    |   movel(p[0.471269, -0.071095, -0.000100, 0.000000, 3.141593, 0.000000],accel_mss,speed_ms,0,blend_radius_m)
    |   movel(p[0.470803, -0.071857, -0.000100, 0.000000, -3.141593, 0.000000],accel_mss,speed_ms,0,blend_radius_m)
    |   movel(p[0.470715, -0.072007, -0.000100, 0.000000, 3.141593, 0.000000],accel_mss,speed_ms,0,0.000)
    |   movel(p[0.470597, -0.072221, -0.000100, 0.000000, -3.141593, 0.000000],accel_mss,speed_ms,0,0.000)
    |   movel(p[0.470473, -0.072456, -0.000100, 0.000000, -3.141593, 0.000000],accel_mss,speed_ms,0,0.000)
    |   movel(p[0.470361, -0.072678, -0.000100, 0.000000, -3.141593, 0.000000],accel_mss,speed_ms,0,0.000)
    |   movel(p[0.470239, -0.072912, -0.000100, 0.000000, -3.141593, 0.000000],accel_mss,speed_ms,0,0.000)
    |   movel(p[0.470084, -0.073181, -0.000100, 0.000000, -3.141593, 0.000000],accel_mss,speed_ms,0,0.000)
    |   movel(p[0.469922, -0.073443, -0.000100, 0.000000, -3.141593, 0.000000],accel_mss,speed_ms,0,0.000)
    |   movel(p[0.469779, -0.073653, -0.000100, 0.000000, -3.141593, 0.000000],accel_mss,speed_ms,0,0.000)
    |   movel(p[0.469648, -0.073842, -0.000100, 0.000000, -3.141593, 0.000000],accel_mss,speed_ms,0,0.000)
    |   movel(p[0.469521, -0.074037, -0.000100, 0.000000, -3.141593, 0.000000],accel_mss,speed_ms,0,0.000)
    |   movel(p[0.469416, -0.074212, -0.000100, 0.000000, -3.141593, 0.000000],accel_mss,speed_ms,0,0.000)
    |   movel(p[0.469356, -0.074328, -0.000100, 0.000000, -3.141593, 0.000000],accel_mss,speed_ms,0,0.000)
    |   movel(p[0.469299, -0.074444, -0.000100, 0.000000, -3.141593, 0.000000],accel_mss,speed_ms,0,0.000)
    |   movel(p[0.469200, -0.074619, -0.000100, 0.000000, -3.141593, 0.000000],accel_mss,speed_ms,0,0.000)
    |   movel(p[0.469084, -0.074815, -0.000100, 0.000000, -3.141593, 0.000000],accel_mss,speed_ms,0,0.000)
    |   movel(p[0.468964, -0.075003, -0.000100, 0.000000, -3.141593, 0.000000],accel_mss,speed_ms,0,0.000)
    |   movel(p[0.468837, -0.075208, -0.000100, 0.000000, -3.141593, 0.000000],accel_mss,speed_ms,0,0.000)
    |   movel(p[0.468696, -0.075453, -0.000100, 0.000000, -3.141593, 0.000000],accel_mss,speed_ms,0,0.000)
    |   movel(p[0.468564, -0.075699, -0.000100, 0.000000, -3.141593, 0.000000],accel_mss,speed_ms,0,0.000)
    |   movel(p[0.468464, -0.075903, -0.000100, 0.000000, -3.141593, 0.000000],accel_mss,speed_ms,0,0.000)
    |   movel(p[0.468366, -0.076091, -0.000100, 0.000000, -3.141593, 0.000000],accel_mss,speed_ms,0,0.000)
    |   movel(p[0.468243, -0.076283, -0.000100, 0.000000, -3.141593, 0.000000],accel_mss,speed_ms,0,0.000)
    |   movel(p[0.468114, -0.076453, -0.000100, 0.000000, 3.141593, 0.000000],accel_mss,speed_ms,0,0.000)
    |   movel(p[0.468002, -0.076565, -0.000100, 0.000000, -3.141593, 0.000000],accel_mss,speed_ms,0,0.000)
    |   movel(p[0.467885, -0.076688, -0.000100, 0.000000, -3.141593, 0.000000],accel_mss,speed_ms,0,0.000)
    |   movel(p[0.467739, -0.076896, -0.000100, 0.000000, -3.141593, 0.000000],accel_mss,speed_ms,0,0.000)
    |   movel(p[0.467592, -0.077142, -0.000100, 0.000000, -3.141593, 0.000000],accel_mss,speed_ms,0,0.000)
    |   movel(p[0.467465, -0.077394, -0.000100, 0.000000, -3.141593, 0.000000],accel_mss,speed_ms,0,0.000)
    |   movel(p[0.467335, -0.077651, -0.000100, 0.000000, -3.141593, 0.000000],accel_mss,speed_ms,0,0.000)
    |   movel(p[0.467175, -0.077912, -0.000100, 0.000000, -3.141593, 0.000000],accel_mss,speed_ms,0,0.000)
    |   movel(p[0.467012, -0.078142, -0.000100, 0.000000, -3.141593, 0.000000],accel_mss,speed_ms,0,0.000)
    |   movel(p[0.466873, -0.078293, -0.000100, 0.000000, -3.141593, 0.000000],accel_mss,speed_ms,0,0.000)
    |   movel(p[0.466753, -0.078412, -0.000100, 0.000000, -3.141593, 0.000000],accel_mss,speed_ms,0,0.000)
    |   movel(p[0.466653, -0.078535, -0.000100, 0.000000, -3.141593, 0.000000],accel_mss,speed_ms,0,0.000)
    |   movel(p[0.466581, -0.078648, -0.000100, 0.000000, -3.141593, 0.000000],accel_mss,speed_ms,0,0.000)
    |   movel(p[0.466531, -0.078815, -0.000100, 0.000000, -3.141593, 0.000000],accel_mss,speed_ms,0,0.000)
    |   movel(p[0.466319, -0.079103, -0.000100, 0.000000, -3.141593, 0.000000],accel_mss,speed_ms,0,0.000)
    |   movel(p[0.466052, -0.079439, -0.000100, 0.000000, -3.141593, 0.000000],accel_mss,speed_ms,0,0.000)
    |   movel(p[0.465736, -0.079810, -0.000100, 0.000000, -3.141593, 0.000000],accel_mss,speed_ms,0,0.000)
    |   movel(p[0.465420, -0.080180, -0.000100, 0.000000, -3.141593, 0.000000],accel_mss,speed_ms,0,0.000)
    |   movel(p[0.465153, -0.080514, -0.000100, 0.000000, -3.141593, 0.000000],accel_mss,speed_ms,0,0.000)
    |   movel(p[0.464939, -0.080799, -0.000100, 0.000000, -3.141593, 0.000000],accel_mss,speed_ms,0,0.000)
    |   movel(p[0.464837, -0.081062, -0.000100, 0.000000, -3.141593, 0.000000],accel_mss,speed_ms,0,0.000)
    |   movel(p[0.464374, -0.081495, -0.000100, 0.000000, 3.141593, 0.000000],accel_mss,speed_ms,0,blend_radius_m)
    |   movel(p[0.463896, -0.081907, -0.000100, 0.000000, -3.141593, 0.000000],accel_mss,speed_ms,0,blend_radius_m)
    |   movel(p[0.463697, -0.081978, -0.000100, 0.000000, -3.141593, 0.000000],accel_mss,speed_ms,0,0.000)
    |   movel(p[0.463600, -0.082033, -0.000100, 0.000000, -3.141593, 0.000000],accel_mss,speed_ms,0,0.000)
    |   movel(p[0.463560, -0.082166, -0.000100, 0.000000, -3.141593, 0.000000],accel_mss,speed_ms,0,0.000)
    |   movel(p[0.463460, -0.082347, -0.000100, 0.000000, -3.141593, 0.000000],accel_mss,speed_ms,0,0.000)
    |   movel(p[0.463351, -0.082441, -0.000100, 0.000000, -3.141593, 0.000000],accel_mss,speed_ms,0,0.000)
    |   movel(p[0.463222, -0.082518, -0.000100, 0.000000, -3.141593, 0.000000],accel_mss,speed_ms,0,0.000)
    |   movel(p[0.463052, -0.082603, -0.000100, 0.000000, -3.141593, 0.000000],accel_mss,speed_ms,0,0.000)
    |   movel(p[0.462809, -0.082727, -0.000100, 0.000000, -3.141593, 0.000000],accel_mss,speed_ms,0,0.000)
    |   movel(p[0.462540, -0.082865, -0.000100, 0.000000, -3.141593, 0.000000],accel_mss,speed_ms,0,0.000)
    |   movel(p[0.462286, -0.082998, -0.000100, 0.000000, -3.141593, 0.000000],accel_mss,speed_ms,0,0.000)
    |   movel(p[0.460770, -0.083741, -0.000100, 0.000000, -3.141593, 0.000000],accel_mss,speed_ms,0,blend_radius_m)
    |   movel(p[0.459479, -0.084259, -0.000100, 0.000000, -3.141593, 0.000000],accel_mss,speed_ms,0,blend_radius_m)
    |   movel(p[0.458369, -0.084574, -0.000100, 0.000000, -3.141593, 0.000000],accel_mss,speed_ms,0,blend_radius_m)
    |   movel(p[0.457411, -0.084692, -0.000100, 0.000000, -3.141593, 0.000000],accel_mss,speed_ms,0,blend_radius_m)
    |   movel(p[0.457160, -0.084702, -0.000100, 0.000000, -3.141593, 0.000000],accel_mss,speed_ms,0,0.000)
    |   movel(p[0.456832, -0.084723, -0.000100, 0.000000, -3.141593, 0.000000],accel_mss,speed_ms,0,0.000)
    |   movel(p[0.456488, -0.084750, -0.000100, 0.000000, -3.141593, 0.000000],accel_mss,speed_ms,0,0.000)
    |   movel(p[0.456178, -0.084780, -0.000100, 0.000000, -3.141593, 0.000000],accel_mss,speed_ms,0,0.000)
    |   movel(p[0.455825, -0.084817, -0.000100, 0.000000, -3.141593, 0.000000],accel_mss,speed_ms,0,0.000)
    |   movel(p[0.455471, -0.084855, -0.000100, 0.000000, -3.141593, 0.000000],accel_mss,speed_ms,0,0.000)
    |   movel(p[0.455487, -0.085515, -0.000100, 0.000000, -3.141593, 0.000000],accel_mss,speed_ms,0,blend_radius_m)
    |   movel(p[0.455503, -0.086174, -0.000100, 0.000000, -3.141593, 0.000000],accel_mss,speed_ms,0,blend_radius_m)
    |   movel(p[0.455510, -0.086885, -0.000100, 0.000000, -3.141593, 0.000000],accel_mss,speed_ms,0,blend_radius_m)
    |   movel(p[0.455478, -0.087299, -0.000100, 0.000000, -3.141593, 0.000000],accel_mss,speed_ms,0,0.000)
    |   movel(p[0.455402, -0.087577, -0.000100, 0.000000, 3.141593, 0.000000],accel_mss,speed_ms,0,0.000)
    |   movel(p[0.455266, -0.087793, -0.000100, 0.000000, -3.141593, 0.000000],accel_mss,speed_ms,0,0.000)
    |   movel(p[0.454617, -0.088208, -0.000100, 0.000000, -3.141593, 0.000000],accel_mss,speed_ms,0,blend_radius_m)
    |   movel(p[0.453609, -0.088391, -0.000100, 0.000000, -3.141593, 0.000000],accel_mss,speed_ms,0,blend_radius_m)
    |   movel(p[0.452601, -0.088329, -0.000100, 0.000000, -3.141593, 0.000000],accel_mss,speed_ms,0,blend_radius_m)
    |   movel(p[0.451957, -0.087990, -0.000100, 0.000000, -3.141593, 0.000000],accel_mss,speed_ms,0,blend_radius_m)
    |   movel(p[0.451797, -0.087787, -0.000100, 0.000000, -3.141593, 0.000000],accel_mss,speed_ms,0,0.000)
    |   movel(p[0.451704, -0.087566, -0.000100, 0.000000, -3.141593, 0.000000],accel_mss,speed_ms,0,0.000)
    |   movel(p[0.451660, -0.087274, -0.000100, 0.000000, -3.141593, 0.000000],accel_mss,speed_ms,0,0.000)
    |   movel(p[0.451656, -0.086831, -0.000100, 0.000000, -3.141593, 0.000000],accel_mss,speed_ms,0,0.000)
    |   movel(p[0.451685, -0.086359, -0.000100, 0.000000, -3.141593, 0.000000],accel_mss,speed_ms,0,0.000)
    |   movel(p[0.451754, -0.086060, -0.000100, 0.000000, -3.141593, 0.000000],accel_mss,speed_ms,0,0.000)
    |   movel(p[0.451891, -0.085814, -0.000100, 0.000000, -3.141593, 0.000000],accel_mss,speed_ms,0,0.000)
    |   movel(p[0.452139, -0.085531, -0.000100, 0.000000, -3.141593, 0.000000],accel_mss,speed_ms,0,0.000)
    |   movel(p[0.452370, -0.085300, -0.000100, 0.000000, -3.141593, 0.000000],accel_mss,speed_ms,0,0.000)
    |   movel(p[0.452601, -0.085069, -0.000100, 0.000000, -3.141593, 0.000000],accel_mss,speed_ms,0,0.000)
    |   movel(p[0.452594, -0.085421, -0.000100, 0.000000, -3.141593, 0.000000],accel_mss,speed_ms,0,0.000)
    |   movel(p[0.452587, -0.085773, -0.000100, 0.000000, -3.141593, 0.000000],accel_mss,speed_ms,0,0.000)
    |   movel(p[0.452617, -0.086277, -0.000100, 0.000000, 3.141593, 0.000000],accel_mss,speed_ms,0,blend_radius_m)
    |   movel(p[0.452736, -0.086636, -0.000100, 0.000000, -3.141593, 0.000000],accel_mss,speed_ms,0,0.000)
    |   movel(p[0.452940, -0.086850, -0.000100, 0.000000, -3.141593, 0.000000],accel_mss,speed_ms,0,0.000)
    |   movel(p[0.453221, -0.086928, -0.000100, 0.000000, -3.141593, 0.000000],accel_mss,speed_ms,0,0.000)
    |   movel(p[0.453501, -0.086830, -0.000100, 0.000000, -3.141593, 0.000000],accel_mss,speed_ms,0,0.000)
    |   movel(p[0.453742, -0.086550, -0.000100, 0.000000, -3.141593, 0.000000],accel_mss,speed_ms,0,0.000)
    |   movel(p[0.453906, -0.086136, -0.000100, 0.000000, -3.141593, 0.000000],accel_mss,speed_ms,0,0.000)
    |   movel(p[0.453961, -0.085650, -0.000100, 0.000000, -3.141593, 0.000000],accel_mss,speed_ms,0,0.000)
    |   movel(p[0.453921, -0.085195, -0.000100, 0.000000, -3.141593, 0.000000],accel_mss,speed_ms,0,0.000)
    |   movel(p[0.453793, -0.084901, -0.000100, 0.000000, -3.141593, 0.000000],accel_mss,speed_ms,0,0.000)
    |   movel(p[0.453566, -0.084736, -0.000100, 0.000000, -3.141593, 0.000000],accel_mss,speed_ms,0,0.000)
    |   movel(p[0.453228, -0.084678, -0.000100, 0.000000, -3.141593, 0.000000],accel_mss,speed_ms,0,0.000)
    |   movel(p[0.452761, -0.084607, -0.000100, 0.000000, -3.141593, 0.000000],accel_mss,speed_ms,0,0.000)
    |   movel(p[0.451120, -0.084082, -0.000100, 0.000000, -3.141593, 0.000000],accel_mss,speed_ms,0,blend_radius_m)
    |   movel(p[0.449478, -0.083535, -0.000100, 0.000000, -3.141593, 0.000000],accel_mss,speed_ms,0,blend_radius_m)
    |   movel(p[0.449086, -0.083326, -0.000100, 0.000000, -3.141593, 0.000000],accel_mss,speed_ms,0,0.000)
    |   movel(p[0.448884, -0.083190, -0.000100, 0.000000, -3.141593, 0.000000],accel_mss,speed_ms,0,0.000)
    |   movel(p[0.448382, -0.082901, -0.000100, 0.000000, -3.141593, 0.000000],accel_mss,speed_ms,0,blend_radius_m)
    |   movel(p[0.447798, -0.082577, -0.000100, 0.000000, -3.141593, 0.000000],accel_mss,speed_ms,0,blend_radius_m)
    |   movel(p[0.447201, -0.082257, -0.000100, 0.000000, 3.141593, 0.000000],accel_mss,speed_ms,0,blend_radius_m)
    |   movel(p[0.446964, -0.082117, -0.000100, 0.000000, -3.141593, 0.000000],accel_mss,speed_ms,0,0.000)
    |   movel(p[0.446696, -0.081927, -0.000100, 0.000000, -3.141593, 0.000000],accel_mss,speed_ms,0,0.000)
    |   movel(p[0.446438, -0.081720, -0.000100, 0.000000, -3.141593, 0.000000],accel_mss,speed_ms,0,0.000)
    |   movel(p[0.446235, -0.081527, -0.000100, 0.000000, -3.141593, 0.000000],accel_mss,speed_ms,0,0.000)
    |   movel(p[0.446056, -0.081355, -0.000100, 0.000000, -3.141593, 0.000000],accel_mss,speed_ms,0,0.000)
    |   movel(p[0.445873, -0.081210, -0.000100, 0.000000, -3.141593, 0.000000],accel_mss,speed_ms,0,0.000)
    |   movel(p[0.445710, -0.081106, -0.000100, 0.000000, -3.141593, 0.000000],accel_mss,speed_ms,0,0.000)
    |   movel(p[0.445608, -0.081078, -0.000100, 0.000000, 3.141593, 0.000000],accel_mss,speed_ms,0,0.000)
    |   movel(p[0.445469, -0.081011, -0.000100, 0.000000, -3.141593, 0.000000],accel_mss,speed_ms,0,0.000)
    |   movel(p[0.445411, -0.080849, -0.000100, 0.000000, -3.141593, 0.000000],accel_mss,speed_ms,0,0.000)
    |   movel(p[0.445334, -0.080659, -0.000100, 0.000000, -3.141593, 0.000000],accel_mss,speed_ms,0,0.000)
    |   movel(p[0.445249, -0.080578, -0.000100, 0.000000, -3.141593, 0.000000],accel_mss,speed_ms,0,0.000)
    |   movel(p[0.445148, -0.080525, -0.000100, 0.000000, -3.141593, 0.000000],accel_mss,speed_ms,0,0.000)
    |   movel(p[0.444857, -0.080365, -0.000100, 0.000000, -3.141593, 0.000000],accel_mss,speed_ms,0,0.000)
    |   movel(p[0.444481, -0.080040, -0.000100, 0.000000, -3.141593, 0.000000],accel_mss,speed_ms,0,0.000)
    |   movel(p[0.444144, -0.079691, -0.000100, 0.000000, -3.141593, 0.000000],accel_mss,speed_ms,0,0.000)
    |   movel(p[0.444065, -0.079492, -0.000100, 0.000000, -3.141593, 0.000000],accel_mss,speed_ms,0,0.000)
    |   movel(p[0.443947, -0.079271, -0.000100, 0.000000, 3.141593, 0.000000],accel_mss,speed_ms,0,0.000)
    |   movel(p[0.443820, -0.079118, -0.000100, 0.000000, -3.141593, 0.000000],accel_mss,speed_ms,0,0.000)
    |   movel(p[0.443670, -0.078967, -0.000100, 0.000000, 3.141593, 0.000000],accel_mss,speed_ms,0,0.000)
    |   movel(p[0.443510, -0.078806, -0.000100, 0.000000, -3.141593, 0.000000],accel_mss,speed_ms,0,0.000)
    |   movel(p[0.443354, -0.078622, -0.000100, 0.000000, 3.141593, 0.000000],accel_mss,speed_ms,0,0.000)
    |   movel(p[0.443222, -0.078444, -0.000100, 0.000000, -3.141593, 0.000000],accel_mss,speed_ms,0,0.000)
    |   movel(p[0.443143, -0.078303, -0.000100, 0.000000, 3.141593, 0.000000],accel_mss,speed_ms,0,0.000)
    |   movel(p[0.443060, -0.078131, -0.000100, 0.000000, -3.141593, 0.000000],accel_mss,speed_ms,0,0.000)
    |   movel(p[0.442893, -0.077805, -0.000100, 0.000000, -3.141593, 0.000000],accel_mss,speed_ms,0,0.000)
    |   movel(p[0.442694, -0.077424, -0.000100, 0.000000, -3.141593, 0.000000],accel_mss,speed_ms,0,0.000)
    |   movel(p[0.442484, -0.077028, -0.000100, 0.000000, 3.141593, 0.000000],accel_mss,speed_ms,0,0.000)
    |   movel(p[0.442106, -0.076250, -0.000100, 0.000000, -3.141593, 0.000000],accel_mss,speed_ms,0,blend_radius_m)
    |   movel(p[0.441737, -0.075346, -0.000100, 0.000000, -3.141593, 0.000000],accel_mss,speed_ms,0,blend_radius_m)
    |   movel(p[0.441438, -0.074482, -0.000100, 0.000000, 3.141593, 0.000000],accel_mss,speed_ms,0,blend_radius_m)
    |   movel(p[0.441290, -0.073856, -0.000100, 0.000000, -3.141593, 0.000000],accel_mss,speed_ms,0,blend_radius_m)
    |   movel(p[0.441095, -0.072461, -0.000100, 0.000000, -3.141593, 0.000000],accel_mss,speed_ms,0,blend_radius_m)
    |   movel(p[0.440999, -0.071329, -0.000100, 0.000000, -3.141593, 0.000000],accel_mss,speed_ms,0,blend_radius_m)
    |   movel(p[0.440988, -0.070256, -0.000100, 0.000000, 3.141593, 0.000000],accel_mss,speed_ms,0,blend_radius_m)
    |   movel(p[0.441055, -0.069048, -0.000100, 0.000000, -3.141593, 0.000000],accel_mss,speed_ms,0,blend_radius_m)
    |   movel(p[0.441120, -0.068309, -0.000100, 0.000000, -3.141593, 0.000000],accel_mss,speed_ms,0,blend_radius_m)
    |   movel(p[0.441186, -0.067613, -0.000100, 0.000000, 3.141593, 0.000000],accel_mss,speed_ms,0,blend_radius_m)
    |   movel(p[0.441247, -0.067027, -0.000100, 0.000000, -3.141593, 0.000000],accel_mss,speed_ms,0,blend_radius_m)
    |   movel(p[0.441285, -0.066753, -0.000100, 0.000000, -3.141593, 0.000000],accel_mss,speed_ms,0,0.000)
    |   movel(p[0.441320, -0.066543, -0.000100, 0.000000, -3.141593, 0.000000],accel_mss,speed_ms,0,0.000)
    |   movel(p[0.441364, -0.066281, -0.000100, 0.000000, -3.141593, 0.000000],accel_mss,speed_ms,0,0.000)
    |   movel(p[0.441408, -0.066012, -0.000100, 0.000000, 3.141593, 0.000000],accel_mss,speed_ms,0,0.000)
    |   movel(p[0.441447, -0.065778, -0.000100, 0.000000, -3.141593, 0.000000],accel_mss,speed_ms,0,0.000)
    |   movel(p[0.441556, -0.065265, -0.000100, 0.000000, 3.141593, 0.000000],accel_mss,speed_ms,0,blend_radius_m)
    |   movel(p[0.441750, -0.064582, -0.000100, 0.000000, -3.141593, 0.000000],accel_mss,speed_ms,0,blend_radius_m)
    |   movel(p[0.441982, -0.063877, -0.000100, 0.000000, -3.141593, 0.000000],accel_mss,speed_ms,0,blend_radius_m)
    |   movel(p[0.442212, -0.063281, -0.000100, 0.000000, -3.141593, 0.000000],accel_mss,speed_ms,0,blend_radius_m)
    |   movel(p[0.442288, -0.063093, -0.000100, 0.000000, -3.141593, 0.000000],accel_mss,speed_ms,0,0.000)
    |   movel(p[0.442352, -0.062922, -0.000100, 0.000000, -3.141593, 0.000000],accel_mss,speed_ms,0,0.000)
    |   movel(p[0.442402, -0.062777, -0.000100, 0.000000, -3.141593, 0.000000],accel_mss,speed_ms,0,0.000)
    |   movel(p[0.442467, -0.062473, -0.000100, 0.000000, -3.141593, 0.000000],accel_mss,speed_ms,0,0.000)
    |   movel(p[0.442814, -0.061765, -0.000100, 0.000000, -3.141593, 0.000000],accel_mss,speed_ms,0,blend_radius_m)
    |   movel(p[0.443178, -0.061071, -0.000100, 0.000000, 3.141593, 0.000000],accel_mss,speed_ms,0,blend_radius_m)
    |   movel(p[0.443358, -0.060852, -0.000100, 0.000000, -3.141593, 0.000000],accel_mss,speed_ms,0,0.000)
    |   movel(p[0.443674, -0.060687, -0.000100, 0.000000, -3.141593, 0.000000],accel_mss,speed_ms,0,0.000)
    |   movel(p[0.444303, -0.060542, -0.000100, 0.000000, -3.141593, 0.000000],accel_mss,speed_ms,0,blend_radius_m)
    |   movel(p[0.444942, -0.060444, -0.000100, 0.000000, -3.141593, 0.000000],accel_mss,speed_ms,0,blend_radius_m)
    |   movel(p[0.445156, -0.060516, -0.000100, 0.000000, 3.141593, 0.000000],accel_mss,speed_ms,0,0.000)
    |   movel(p[0.445177, -0.060614, -0.000100, 0.000000, -3.141593, 0.000000],accel_mss,speed_ms,0,0.000)
    |   movel(p[0.444985, -0.061101, -0.000100, 0.000000, -3.141593, 0.000000],accel_mss,speed_ms,0,blend_radius_m)
    |   movel(p[0.444730, -0.061679, -0.000100, 0.000000, -3.141593, 0.000000],accel_mss,speed_ms,0,blend_radius_m)
    |   movel(p[0.444406, -0.062343, -0.000100, 0.000000, -3.141593, 0.000000],accel_mss,speed_ms,0,blend_radius_m)
    |   movel(p[0.443971, -0.063198, -0.000100, 0.000000, 3.141593, 0.000000],accel_mss,speed_ms,0,blend_radius_m)
    |   movel(p[0.443536, -0.064053, -0.000100, 0.000000, -3.141593, 0.000000],accel_mss,speed_ms,0,blend_radius_m)
    |   movel(p[0.443521, -0.065328, -0.000100, 0.000000, -3.141593, 0.000000],accel_mss,speed_ms,0,blend_radius_m)
    |   movel(p[0.443507, -0.066603, -0.000100, 0.000000, -3.141593, 0.000000],accel_mss,speed_ms,0,blend_radius_m)
    |   movel(p[0.443507, -0.067635, -0.000100, 0.000000, 3.141593, 0.000000],accel_mss,speed_ms,0,blend_radius_m)
    |   movel(p[0.443532, -0.068625, -0.000100, 0.000000, 3.141593, 0.000000],accel_mss,speed_ms,0,blend_radius_m)
    |   movel(p[0.443574, -0.069465, -0.000100, 0.000000, -3.141593, 0.000000],accel_mss,speed_ms,0,blend_radius_m)
    |   movel(p[0.443632, -0.069903, -0.000100, 0.000000, 3.141593, 0.000000],accel_mss,speed_ms,0,0.000)
    |   movel(p[0.444078, -0.071666, -0.000100, 0.000000, -3.141593, 0.000000],accel_mss,speed_ms,0,blend_radius_m)
    |   movel(p[0.444658, -0.073264, -0.000100, 0.000000, -3.141593, 0.000000],accel_mss,speed_ms,0,blend_radius_m)
    |   movel(p[0.445338, -0.074619, -0.000100, 0.000000, 3.141593, 0.000000],accel_mss,speed_ms,0,blend_radius_m)
    |   movel(p[0.446084, -0.075645, -0.000100, 0.000000, -3.141593, 0.000000],accel_mss,speed_ms,0,blend_radius_m)
    |   movel(p[0.446343, -0.075942, -0.000100, 0.000000, -3.141593, 0.000000],accel_mss,speed_ms,0,0.000)
    |   movel(p[0.446562, -0.076211, -0.000100, 0.000000, -3.141593, 0.000000],accel_mss,speed_ms,0,0.000)
    |   movel(p[0.446737, -0.076442, -0.000100, 0.000000, -3.141593, 0.000000],accel_mss,speed_ms,0,0.000)
    |   movel(p[0.446821, -0.076682, -0.000100, 0.000000, -3.141593, 0.000000],accel_mss,speed_ms,0,0.000)
    |   movel(p[0.447095, -0.076986, -0.000100, 0.000000, -3.141593, 0.000000],accel_mss,speed_ms,0,0.000)
    |   movel(p[0.447392, -0.077267, -0.000100, 0.000000, -3.141593, 0.000000],accel_mss,speed_ms,0,0.000)
    |   movel(p[0.447554, -0.077328, -0.000100, 0.000000, -3.141593, 0.000000],accel_mss,speed_ms,0,0.000)
    |   movel(p[0.447902, -0.077540, -0.000100, 0.000000, -3.141593, 0.000000],accel_mss,speed_ms,0,0.000)
    |   movel(p[0.448206, -0.077774, -0.000100, 0.000000, -3.141593, 0.000000],accel_mss,speed_ms,0,0.000)
    |   movel(p[0.448541, -0.078051, -0.000100, 0.000000, -3.141593, 0.000000],accel_mss,speed_ms,0,0.000)
    |   movel(p[0.448908, -0.078346, -0.000100, 0.000000, -3.141593, 0.000000],accel_mss,speed_ms,0,0.000)
    |   movel(p[0.449314, -0.078637, -0.000100, 0.000000, -3.141593, 0.000000],accel_mss,speed_ms,0,0.000)
    |   movel(p[0.449697, -0.078884, -0.000100, 0.000000, -3.141593, 0.000000],accel_mss,speed_ms,0,0.000)
    |   movel(p[0.449986, -0.079033, -0.000100, 0.000000, -3.141593, 0.000000],accel_mss,speed_ms,0,0.000)
    |   movel(p[0.450235, -0.079143, -0.000100, 0.000000, -3.141593, 0.000000],accel_mss,speed_ms,0,0.000)
    |   movel(p[0.450487, -0.079258, -0.000100, 0.000000, -3.141593, 0.000000],accel_mss,speed_ms,0,0.000)
    |   movel(p[0.450708, -0.079364, -0.000100, 0.000000, -3.141593, 0.000000],accel_mss,speed_ms,0,0.000)
    |   movel(p[0.450848, -0.079436, -0.000100, 0.000000, -3.141593, 0.000000],accel_mss,speed_ms,0,0.000)
    |   movel(p[0.451298, -0.079673, -0.000100, 0.000000, -3.141593, 0.000000],accel_mss,speed_ms,0,blend_radius_m)
    |   movel(p[0.451639, -0.079837, -0.000100, 0.000000, 3.141593, 0.000000],accel_mss,speed_ms,0,0.000)
    |   movel(p[0.452020, -0.079998, -0.000100, 0.000000, -3.141593, 0.000000],accel_mss,speed_ms,0,0.000)
    |   movel(p[0.452633, -0.080235, -0.000100, 0.000000, -3.141593, 0.000000],accel_mss,speed_ms,0,blend_radius_m)
    |   movel(p[0.454596, -0.080839, -0.000100, 0.000000, -3.141593, 0.000000],accel_mss,speed_ms,0,blend_radius_m)
    |   movel(p[0.456325, -0.081062, -0.000100, 0.000000, -3.141593, 0.000000],accel_mss,speed_ms,0,blend_radius_m)
    |   movel(p[0.458130, -0.080924, -0.000100, 0.000000, -3.141593, 0.000000],accel_mss,speed_ms,0,blend_radius_m)
    |   movel(p[0.460338, -0.080412, -0.000100, 0.000000, -3.141593, 0.000000],accel_mss,speed_ms,0,blend_radius_m)
    |   movel(p[0.461163, -0.080152, -0.000100, 0.000000, -3.141593, 0.000000],accel_mss,speed_ms,0,blend_radius_m)
    |   movel(p[0.461802, -0.079896, -0.000100, 0.000000, -3.141593, 0.000000],accel_mss,speed_ms,0,blend_radius_m)
    |   movel(p[0.462430, -0.079570, -0.000100, 0.000000, -3.141593, 0.000000],accel_mss,speed_ms,0,blend_radius_m)
    |   movel(p[0.463220, -0.079086, -0.000100, 0.000000, -3.141593, 0.000000],accel_mss,speed_ms,0,blend_radius_m)
    |   movel(p[0.463474, -0.078930, -0.000100, 0.000000, -3.141593, 0.000000],accel_mss,speed_ms,0,0.000)
    |   movel(p[0.463709, -0.078798, -0.000100, 0.000000, -3.141593, 0.000000],accel_mss,speed_ms,0,0.000)
    |   movel(p[0.463909, -0.078698, -0.000100, 0.000000, -3.141593, 0.000000],accel_mss,speed_ms,0,0.000)
    |   movel(p[0.464246, -0.078577, -0.000100, 0.000000, -3.141593, 0.000000],accel_mss,speed_ms,0,0.000)
    |   movel(p[0.465145, -0.077696, -0.000100, 0.000000, -3.141593, 0.000000],accel_mss,speed_ms,0,blend_radius_m)
    |   movel(p[0.465988, -0.076825, -0.000100, 0.000000, -3.141593, 0.000000],accel_mss,speed_ms,0,blend_radius_m)
    |   movel(p[0.466257, -0.076416, -0.000100, 0.000000, -3.141593, 0.000000],accel_mss,speed_ms,0,0.000)
    |   movel(p[0.466339, -0.076245, -0.000100, 0.000000, -3.141593, 0.000000],accel_mss,speed_ms,0,0.000)
    |   movel(p[0.466456, -0.076028, -0.000100, 0.000000, -3.141593, 0.000000],accel_mss,speed_ms,0,0.000)
    |   movel(p[0.466587, -0.075802, -0.000100, 0.000000, 3.141593, 0.000000],accel_mss,speed_ms,0,0.000)
    |   movel(p[0.466712, -0.075603, -0.000100, 0.000000, 3.141593, 0.000000],accel_mss,speed_ms,0,0.000)
    |   movel(p[0.466832, -0.075415, -0.000100, 0.000000, -3.141593, 0.000000],accel_mss,speed_ms,0,0.000)
    |   movel(p[0.466951, -0.075219, -0.000100, 0.000000, -3.141593, 0.000000],accel_mss,speed_ms,0,0.000)
    |   movel(p[0.467052, -0.075044, -0.000100, 0.000000, -3.141593, 0.000000],accel_mss,speed_ms,0,0.000)
    |   movel(p[0.467111, -0.074928, -0.000100, 0.000000, -3.141593, 0.000000],accel_mss,speed_ms,0,0.000)
    |   movel(p[0.467171, -0.074812, -0.000100, 0.000000, -3.141593, 0.000000],accel_mss,speed_ms,0,0.000)
    |   movel(p[0.467278, -0.074637, -0.000100, 0.000000, -3.141593, 0.000000],accel_mss,speed_ms,0,0.000)
    |   movel(p[0.467406, -0.074442, -0.000100, 0.000000, -3.141593, 0.000000],accel_mss,speed_ms,0,0.000)
    |   movel(p[0.467537, -0.074253, -0.000100, 0.000000, -3.141593, 0.000000],accel_mss,speed_ms,0,0.000)
    |   movel(p[0.467779, -0.073867, -0.000100, 0.000000, -3.141593, 0.000000],accel_mss,speed_ms,0,0.000)
    |   movel(p[0.468125, -0.073209, -0.000100, 0.000000, -3.141593, 0.000000],accel_mss,speed_ms,0,blend_radius_m)
    |   movel(p[0.468601, -0.072244, -0.000100, 0.000000, -3.141593, 0.000000],accel_mss,speed_ms,0,blend_radius_m)
    |   movel(p[0.469302, -0.070766, -0.000100, 0.000000, -3.141593, 0.000000],accel_mss,speed_ms,0,blend_radius_m)
    |   movel(p[0.469447, -0.070232, -0.000100, 0.000000, -3.141593, 0.000000],accel_mss,speed_ms,0,blend_radius_m)
    |   movel(p[0.469461, -0.069462, -0.000100, 0.000000, -3.141593, 0.000000],accel_mss,speed_ms,0,blend_radius_m)
    |   movel(p[0.469371, -0.068706, -0.000100, 0.000000, -3.141593, 0.000000],accel_mss,speed_ms,0,blend_radius_m)
    |   movel(p[0.469175, -0.068228, -0.000100, 0.000000, -3.141593, 0.000000],accel_mss,speed_ms,0,blend_radius_m)
    |   movel(p[0.469055, -0.068043, -0.000100, 0.000000, -3.141593, 0.000000],accel_mss,speed_ms,0,0.000)
    |   movel(p[0.468928, -0.067841, -0.000100, 0.000000, -3.141593, 0.000000],accel_mss,speed_ms,0,0.000)
    |   movel(p[0.468814, -0.067650, -0.000100, 0.000000, -3.141593, 0.000000],accel_mss,speed_ms,0,0.000)
    |   movel(p[0.468735, -0.067506, -0.000100, 0.000000, -3.141593, 0.000000],accel_mss,speed_ms,0,0.000)
    |   movel(p[0.468653, -0.067381, -0.000100, 0.000000, -3.141593, 0.000000],accel_mss,speed_ms,0,0.000)
    |   movel(p[0.468536, -0.067252, -0.000100, 0.000000, 3.141593, 0.000000],accel_mss,speed_ms,0,0.000)
    |   movel(p[0.468404, -0.067136, -0.000100, 0.000000, -3.141593, 0.000000],accel_mss,speed_ms,0,0.000)
    |   movel(p[0.468276, -0.067056, -0.000100, 0.000000, -3.141593, 0.000000],accel_mss,speed_ms,0,0.000)
    |   movel(p[0.468116, -0.066964, -0.000100, 0.000000, -3.141593, 0.000000],accel_mss,speed_ms,0,0.000)
    |   movel(p[0.467867, -0.066794, -0.000100, 0.000000, -3.141593, 0.000000],accel_mss,speed_ms,0,0.000)
    |   movel(p[0.467586, -0.066591, -0.000100, 0.000000, -3.141593, 0.000000],accel_mss,speed_ms,0,0.000)
    |   movel(p[0.467311, -0.066378, -0.000100, 0.000000, -3.141593, 0.000000],accel_mss,speed_ms,0,0.000)
    |   movel(p[0.466855, -0.066027, -0.000100, 0.000000, -3.141593, 0.000000],accel_mss,speed_ms,0,blend_radius_m)
    |   movel(p[0.466477, -0.065761, -0.000100, 0.000000, -3.141593, 0.000000],accel_mss,speed_ms,0,0.000)
    |   movel(p[0.466139, -0.065555, -0.000100, 0.000000, -3.141593, 0.000000],accel_mss,speed_ms,0,0.000)
    |   movel(p[0.465811, -0.065387, -0.000100, 0.000000, -3.141593, 0.000000],accel_mss,speed_ms,0,0.000)
    |   movel(p[0.464432, -0.064787, -0.000100, 0.000000, -3.141593, 0.000000],accel_mss,speed_ms,0,blend_radius_m)
    |   movel(p[0.463392, -0.064409, -0.000100, 0.000000, -3.141593, 0.000000],accel_mss,speed_ms,0,blend_radius_m)
    |   movel(p[0.462552, -0.064198, -0.000100, 0.000000, -3.141593, 0.000000],accel_mss,speed_ms,0,blend_radius_m)
    |   movel(p[0.461816, -0.064128, -0.000100, 0.000000, -3.141593, 0.000000],accel_mss,speed_ms,0,blend_radius_m)
    |   movel(p[0.461140, -0.064183, -0.000100, 0.000000, -3.141593, 0.000000],accel_mss,speed_ms,0,blend_radius_m)
    |   movel(p[0.460331, -0.064354, -0.000100, 0.000000, -3.141593, 0.000000],accel_mss,speed_ms,0,blend_radius_m)
    |   movel(p[0.459588, -0.064579, -0.000100, 0.000000, 3.141593, 0.000000],accel_mss,speed_ms,0,blend_radius_m)
    |   movel(p[0.459213, -0.064801, -0.000100, 0.000000, -3.141593, 0.000000],accel_mss,speed_ms,0,0.000)
    |   movel(p[0.459107, -0.064888, -0.000100, 0.000000, -3.141593, 0.000000],accel_mss,speed_ms,0,0.000)
    |   movel(p[0.458994, -0.064962, -0.000100, 0.000000, -3.141593, 0.000000],accel_mss,speed_ms,0,0.000)
    |   movel(p[0.458890, -0.065013, -0.000100, 0.000000, -3.141593, 0.000000],accel_mss,speed_ms,0,0.000)
    |   movel(p[0.458612, -0.065112, -0.000100, 0.000000, -3.141593, 0.000000],accel_mss,speed_ms,0,0.000)
    |   movel(p[0.457952, -0.065766, -0.000100, 0.000000, -3.141593, 0.000000],accel_mss,speed_ms,0,blend_radius_m)
    |   movel(p[0.457336, -0.066421, -0.000100, 0.000000, -3.141593, 0.000000],accel_mss,speed_ms,0,blend_radius_m)
    |   movel(p[0.457025, -0.066849, -0.000100, 0.000000, 3.141593, 0.000000],accel_mss,speed_ms,0,blend_radius_m)
    |   movel(p[0.456591, -0.067674, -0.000100, 0.000000, -3.141593, 0.000000],accel_mss,speed_ms,0,blend_radius_m)
    |   movel(p[0.456398, -0.068275, -0.000100, 0.000000, -3.141593, 0.000000],accel_mss,speed_ms,0,blend_radius_m)
    |   movel(p[0.456405, -0.068758, -0.000100, 0.000000, -3.141593, 0.000000],accel_mss,speed_ms,0,0.000)
    |   movel(p[0.456595, -0.069196, -0.000100, 0.000000, -3.141593, 0.000000],accel_mss,speed_ms,0,0.000)
    |   movel(p[0.457221, -0.069718, -0.000100, 0.000000, -3.141593, 0.000000],accel_mss,speed_ms,0,blend_radius_m)
    |   movel(p[0.458229, -0.070037, -0.000100, 0.000000, -3.141593, 0.000000],accel_mss,speed_ms,0,blend_radius_m)
    |   movel(p[0.459323, -0.070098, -0.000100, 0.000000, -3.141593, 0.000000],accel_mss,speed_ms,0,blend_radius_m)
    |   movel(p[0.460213, -0.069853, -0.000100, 0.000000, -3.141593, 0.000000],accel_mss,speed_ms,0,blend_radius_m)
    |   movel(p[0.460475, -0.069701, -0.000100, 0.000000, -3.141593, 0.000000],accel_mss,speed_ms,0,0.000)
    |   movel(p[0.460756, -0.069500, -0.000100, 0.000000, -3.141593, 0.000000],accel_mss,speed_ms,0,0.000)
    |   movel(p[0.461015, -0.069285, -0.000100, 0.000000, -3.141593, 0.000000],accel_mss,speed_ms,0,0.000)
    |   movel(p[0.461204, -0.069089, -0.000100, 0.000000, 3.141593, 0.000000],accel_mss,speed_ms,0,0.000)
    |   movel(p[0.461465, -0.068715, -0.000100, 0.000000, -3.141593, 0.000000],accel_mss,speed_ms,0,0.000)
    |   movel(p[0.461706, -0.068232, -0.000100, 0.000000, -3.141593, 0.000000],accel_mss,speed_ms,0,blend_radius_m)
    |   movel(p[0.461881, -0.067764, -0.000100, 0.000000, -3.141593, 0.000000],accel_mss,speed_ms,0,0.000)
    |   movel(p[0.461899, -0.067483, -0.000100, 0.000000, -3.141593, 0.000000],accel_mss,speed_ms,0,0.000)
    |   movel(p[0.461864, -0.067205, -0.000100, 0.000000, -3.141593, 0.000000],accel_mss,speed_ms,0,0.000)
    |   movel(p[0.461916, -0.067104, -0.000100, 0.000000, -3.141593, 0.000000],accel_mss,speed_ms,0,0.000)
    |   movel(p[0.462137, -0.067333, -0.000100, 0.000000, -3.141593, 0.000000],accel_mss,speed_ms,0,0.000)
    |   movel(p[0.462346, -0.068412, -0.000100, 0.000000, -3.141593, 0.000000],accel_mss,speed_ms,0,blend_radius_m)
    |   movel(p[0.461970, -0.069582, -0.000100, 0.000000, -3.141593, 0.000000],accel_mss,speed_ms,0,blend_radius_m)
    |   movel(p[0.461091, -0.070600, -0.000100, 0.000000, -3.141593, 0.000000],accel_mss,speed_ms,0,blend_radius_m)
    |   movel(p[0.459886, -0.071238, -0.000100, 0.000000, -3.141593, 0.000000],accel_mss,speed_ms,0,blend_radius_m)
    |   movel(p[0.457985, -0.071527, -0.000100, 0.000000, -3.141593, 0.000000],accel_mss,speed_ms,0,blend_radius_m)
    |   movel(p[0.456249, -0.071174, -0.000100, 0.000000, -3.141593, 0.000000],accel_mss,speed_ms,0,blend_radius_m)
    |   movel(p[0.454948, -0.070242, -0.000100, 0.000000, -3.141593, 0.000000],accel_mss,speed_ms,0,blend_radius_m)
    |   movel(p[0.454267, -0.068884, -0.000100, 0.000000, -3.141593, 0.000000],accel_mss,speed_ms,0,blend_radius_m)
    |   movel(p[0.454212, -0.067480, -0.000100, 0.000000, -3.141593, 0.000000],accel_mss,speed_ms,0,blend_radius_m)
    |   movel(p[0.454596, -0.065987, -0.000100, 0.000000, -3.141593, 0.000000],accel_mss,speed_ms,0,blend_radius_m)
    |   movel(p[0.455391, -0.064501, -0.000100, 0.000000, 3.141593, 0.000000],accel_mss,speed_ms,0,blend_radius_m)
    |   movel(p[0.456551, -0.063122, -0.000100, 0.000000, -3.141593, 0.000000],accel_mss,speed_ms,0,blend_radius_m)
    |   movel(p[0.457269, -0.062447, -0.000100, 0.000000, -3.141593, 0.000000],accel_mss,speed_ms,0,blend_radius_m)
    |   movel(p[0.457874, -0.061954, -0.000100, 0.000000, -3.141593, 0.000000],accel_mss,speed_ms,0,blend_radius_m)
    |   movel(p[0.458444, -0.061579, -0.000100, 0.000000, 3.141593, 0.000000],accel_mss,speed_ms,0,blend_radius_m)
    |   movel(p[0.459048, -0.061275, -0.000100, 0.000000, -3.141593, 0.000000],accel_mss,speed_ms,0,blend_radius_m)
    |   movel(p[0.459216, -0.061190, -0.000100, 0.000000, -3.141593, 0.000000],accel_mss,speed_ms,0,0.000)
    |   movel(p[0.459292, -0.061114, -0.000100, 0.000000, -3.141593, 0.000000],accel_mss,speed_ms,0,0.000)
    |   movel(p[0.459240, -0.060947, -0.000100, 0.000000, 3.141593, 0.000000],accel_mss,speed_ms,0,0.000)
    |   movel(p[0.459222, -0.060794, -0.000100, 0.000000, -3.141593, 0.000000],accel_mss,speed_ms,0,0.000)
    |   movel(p[0.459469, -0.060442, -0.000100, 0.000000, -3.141593, 0.000000],accel_mss,speed_ms,0,0.000)
    |   movel(p[0.459918, -0.059918, -0.000100, 0.000000, -3.141593, 0.000000],accel_mss,speed_ms,0,blend_radius_m)
    |   movel(p[0.460708, -0.059087, -0.000100, 0.000000, -3.141593, 0.000000],accel_mss,speed_ms,0,blend_radius_m)
    |   movel(p[0.461630, -0.058085, -0.000100, 0.000000, -3.141593, 0.000000],accel_mss,speed_ms,0,blend_radius_m)
    |   movel(p[0.462326, -0.057213, -0.000100, 0.000000, -3.141593, 0.000000],accel_mss,speed_ms,0,blend_radius_m)
    |   movel(p[0.462806, -0.056470, -0.000100, 0.000000, -3.141593, 0.000000],accel_mss,speed_ms,0,blend_radius_m)
    |   movel(p[0.463039, -0.055878, -0.000100, 0.000000, -3.141593, 0.000000],accel_mss,speed_ms,0,blend_radius_m)
    |   movel(p[0.463164, -0.055583, -0.000100, 0.000000, -3.141593, 0.000000],accel_mss,speed_ms,0,0.000)
    |   movel(p[0.463292, -0.055300, -0.000100, 0.000000, -3.141593, 0.000000],accel_mss,speed_ms,0,0.000)
    |   movel(p[0.463440, -0.054978, -0.000100, 0.000000, -3.141593, 0.000000],accel_mss,speed_ms,0,0.000)
    |   movel(p[0.463814, -0.054136, -0.000100, 0.000000, -3.141593, 0.000000],accel_mss,speed_ms,0,blend_radius_m)
    |   movel(p[0.464034, -0.053528, -0.000100, 0.000000, -3.141593, 0.000000],accel_mss,speed_ms,0,blend_radius_m)
    |   movel(p[0.464136, -0.053085, -0.000100, 0.000000, -3.141593, 0.000000],accel_mss,speed_ms,0,0.000)
    |   movel(p[0.464106, -0.052802, -0.000100, 0.000000, -3.141593, 0.000000],accel_mss,speed_ms,0,0.000)
    |   movel(p[0.464038, -0.052653, -0.000100, 0.000000, -3.141593, 0.000000],accel_mss,speed_ms,0,0.000)
    |   movel(p[0.463901, -0.052640, -0.000100, 0.000000, -3.141593, 0.000000],accel_mss,speed_ms,0,0.000)
    |   movel(p[0.463734, -0.052783, -0.000100, 0.000000, -3.141593, 0.000000],accel_mss,speed_ms,0,0.000)
    |   movel(p[0.463619, -0.052877, -0.000100, 0.000000, -3.141593, 0.000000],accel_mss,speed_ms,0,0.000)
    |   movel(p[0.463499, -0.052956, -0.000100, 0.000000, 3.141593, 0.000000],accel_mss,speed_ms,0,0.000)
    |   movel(p[0.463390, -0.053012, -0.000100, 0.000000, -3.141593, 0.000000],accel_mss,speed_ms,0,0.000)
    |   movel(p[0.463233, -0.053055, -0.000100, 0.000000, -3.141593, 0.000000],accel_mss,speed_ms,0,0.000)
    |   movel(p[0.463063, -0.053183, -0.000100, 0.000000, -3.141593, 0.000000],accel_mss,speed_ms,0,0.000)
    |   movel(p[0.462867, -0.053352, -0.000100, 0.000000, -3.141593, 0.000000],accel_mss,speed_ms,0,0.000)
    |   movel(p[0.462661, -0.053553, -0.000100, 0.000000, -3.141593, 0.000000],accel_mss,speed_ms,0,0.000)
    |   movel(p[0.462456, -0.053754, -0.000100, 0.000000, -3.141593, 0.000000],accel_mss,speed_ms,0,0.000)
    |   movel(p[0.462259, -0.053924, -0.000100, 0.000000, -3.141593, 0.000000],accel_mss,speed_ms,0,0.000)
    |   movel(p[0.462090, -0.054052, -0.000100, 0.000000, -3.141593, 0.000000],accel_mss,speed_ms,0,0.000)
    |   movel(p[0.461927, -0.054097, -0.000100, 0.000000, -3.141593, 0.000000],accel_mss,speed_ms,0,0.000)
    |   movel(p[0.461770, -0.054180, -0.000100, 0.000000, -3.141593, 0.000000],accel_mss,speed_ms,0,0.000)
    |   movel(p[0.461588, -0.054292, -0.000100, 0.000000, -3.141593, 0.000000],accel_mss,speed_ms,0,0.000)
    |   movel(p[0.461400, -0.054424, -0.000100, 0.000000, -3.141593, 0.000000],accel_mss,speed_ms,0,0.000)
    |   movel(p[0.460997, -0.054688, -0.000100, 0.000000, -3.141593, 0.000000],accel_mss,speed_ms,0,0.000)
    |   movel(p[0.460404, -0.055008, -0.000100, 0.000000, -3.141593, 0.000000],accel_mss,speed_ms,0,blend_radius_m)
    |   movel(p[0.459658, -0.055372, -0.000100, 0.000000, -3.141593, 0.000000],accel_mss,speed_ms,0,blend_radius_m)
    |   movel(p[0.458761, -0.055774, -0.000100, 0.000000, -3.141593, 0.000000],accel_mss,speed_ms,0,blend_radius_m)
    |   movel(p[0.458517, -0.055868, -0.000100, 0.000000, -3.141593, 0.000000],accel_mss,speed_ms,0,0.000)
    |   movel(p[0.458214, -0.055963, -0.000100, 0.000000, -3.141593, 0.000000],accel_mss,speed_ms,0,0.000)
    |   movel(p[0.457904, -0.056045, -0.000100, 0.000000, -3.141593, 0.000000],accel_mss,speed_ms,0,0.000)
    |   movel(p[0.457636, -0.056098, -0.000100, 0.000000, -3.141593, 0.000000],accel_mss,speed_ms,0,0.000)
    |   movel(p[0.457384, -0.056141, -0.000100, 0.000000, -3.141593, 0.000000],accel_mss,speed_ms,0,0.000)
    |   movel(p[0.457124, -0.056191, -0.000100, 0.000000, -3.141593, 0.000000],accel_mss,speed_ms,0,0.000)
    |   movel(p[0.456891, -0.056241, -0.000100, 0.000000, 3.141593, 0.000000],accel_mss,speed_ms,0,0.000)
    |   movel(p[0.456736, -0.056280, -0.000100, 0.000000, 3.141593, 0.000000],accel_mss,speed_ms,0,0.000)
    |   movel(p[0.456571, -0.056318, -0.000100, 0.000000, 3.141593, 0.000000],accel_mss,speed_ms,0,0.000)
    |   movel(p[0.456580, -0.056214, -0.000100, 0.000000, -3.141593, 0.000000],accel_mss,speed_ms,0,0.000)
    |   movel(p[0.456800, -0.055972, -0.000100, 0.000000, -3.141593, 0.000000],accel_mss,speed_ms,0,0.000)
    |   movel(p[0.456951, -0.055821, -0.000100, 0.000000, -3.141593, 0.000000],accel_mss,speed_ms,0,0.000)
    |   movel(p[0.457104, -0.055693, -0.000100, 0.000000, -3.141593, 0.000000],accel_mss,speed_ms,0,0.000)
    |   movel(p[0.457240, -0.055601, -0.000100, 0.000000, -3.141593, 0.000000],accel_mss,speed_ms,0,0.000)
    |   movel(p[0.457427, -0.055540, -0.000100, 0.000000, -3.141593, 0.000000],accel_mss,speed_ms,0,0.000)
    |   movel(p[0.457791, -0.055250, -0.000100, 0.000000, -3.141593, 0.000000],accel_mss,speed_ms,0,0.000)
    |   movel(p[0.458214, -0.054893, -0.000100, 0.000000, -3.141593, 0.000000],accel_mss,speed_ms,0,blend_radius_m)
    |   movel(p[0.458686, -0.054470, -0.000100, 0.000000, -3.141593, 0.000000],accel_mss,speed_ms,0,blend_radius_m)
    |   movel(p[0.459286, -0.053917, -0.000100, 0.000000, -3.141593, 0.000000],accel_mss,speed_ms,0,blend_radius_m)
    |   movel(p[0.459886, -0.053365, -0.000100, 0.000000, -3.141593, 0.000000],accel_mss,speed_ms,0,blend_radius_m)
    |   movel(p[0.459698, -0.053203, -0.000100, 0.000000, -3.141593, 0.000000],accel_mss,speed_ms,0,0.000)
    |   movel(p[0.459511, -0.053041, -0.000100, 0.000000, -3.141593, 0.000000],accel_mss,speed_ms,0,0.000)
    |   movel(p[0.459343, -0.052907, -0.000100, 0.000000, -3.141593, 0.000000],accel_mss,speed_ms,0,0.000)
    |   movel(p[0.459147, -0.052771, -0.000100, 0.000000, -3.141593, 0.000000],accel_mss,speed_ms,0,0.000)
    |   movel(p[0.458954, -0.052654, -0.000100, 0.000000, 3.141593, 0.000000],accel_mss,speed_ms,0,0.000)
    |   movel(p[0.458798, -0.052577, -0.000100, 0.000000, -3.141593, 0.000000],accel_mss,speed_ms,0,0.000)
    |   movel(p[0.458585, -0.052395, -0.000100, 0.000000, -3.141593, 0.000000],accel_mss,speed_ms,0,0.000)
    |   movel(p[0.458467, -0.052084, -0.000100, 0.000000, -3.141593, 0.000000],accel_mss,speed_ms,0,0.000)
    |   movel(p[0.458470, -0.051722, -0.000100, 0.000000, -3.141593, 0.000000],accel_mss,speed_ms,0,0.000)
    |   movel(p[0.458598, -0.051394, -0.000100, 0.000000, 3.141593, 0.000000],accel_mss,speed_ms,0,0.000)
    |   movel(p[0.458723, -0.051287, -0.000100, 0.000000, 3.141593, 0.000000],accel_mss,speed_ms,0,0.000)
    |   movel(p[0.458878, -0.051277, -0.000100, 0.000000, -3.141593, 0.000000],accel_mss,speed_ms,0,0.000)
    |   movel(p[0.459118, -0.051382, -0.000100, 0.000000, -3.141593, 0.000000],accel_mss,speed_ms,0,0.000)
    |   movel(p[0.459586, -0.051678, -0.000100, 0.000000, 3.141593, 0.000000],accel_mss,speed_ms,0,blend_radius_m)
    |   movel(p[0.459780, -0.051802, -0.000100, 0.000000, -3.141593, 0.000000],accel_mss,speed_ms,0,0.000)
    |   movel(p[0.459992, -0.051932, -0.000100, 0.000000, 3.141593, 0.000000],accel_mss,speed_ms,0,0.000)
    |   movel(p[0.460190, -0.052047, -0.000100, 0.000000, 3.141593, 0.000000],accel_mss,speed_ms,0,0.000)
    |   movel(p[0.460336, -0.052126, -0.000100, 0.000000, -3.141593, 0.000000],accel_mss,speed_ms,0,0.000)
    |   movel(p[0.460469, -0.052197, -0.000100, 0.000000, -3.141593, 0.000000],accel_mss,speed_ms,0,0.000)
    |   movel(p[0.460623, -0.052287, -0.000100, 0.000000, 3.141593, 0.000000],accel_mss,speed_ms,0,0.000)
    |   movel(p[0.460773, -0.052380, -0.000100, 0.000000, -3.141593, 0.000000],accel_mss,speed_ms,0,0.000)
    |   movel(p[0.460893, -0.052461, -0.000100, 0.000000, -3.141593, 0.000000],accel_mss,speed_ms,0,0.000)
    |   movel(p[0.461045, -0.052537, -0.000100, 0.000000, -3.141593, 0.000000],accel_mss,speed_ms,0,0.000)
    |   movel(p[0.461180, -0.052538, -0.000100, 0.000000, -3.141593, 0.000000],accel_mss,speed_ms,0,0.000)
    |   movel(p[0.461334, -0.052457, -0.000100, 0.000000, -3.141593, 0.000000],accel_mss,speed_ms,0,0.000)
    |   movel(p[0.461568, -0.052255, -0.000100, 0.000000, -3.141593, 0.000000],accel_mss,speed_ms,0,0.000)
    |   movel(p[0.461741, -0.052102, -0.000100, 0.000000, -3.141593, 0.000000],accel_mss,speed_ms,0,0.000)
    |   movel(p[0.461915, -0.051964, -0.000100, 0.000000, 3.141593, 0.000000],accel_mss,speed_ms,0,0.000)
    |   movel(p[0.462068, -0.051855, -0.000100, 0.000000, -3.141593, 0.000000],accel_mss,speed_ms,0,0.000)
    |   movel(p[0.462162, -0.051810, -0.000100, 0.000000, -3.141593, 0.000000],accel_mss,speed_ms,0,0.000)
    |   movel(p[0.462275, -0.051749, -0.000100, 0.000000, -3.141593, 0.000000],accel_mss,speed_ms,0,0.000)
    |   movel(p[0.462675, -0.051431, -0.000100, 0.000000, -3.141593, 0.000000],accel_mss,speed_ms,0,blend_radius_m)
    |   movel(p[0.463141, -0.051046, -0.000100, 0.000000, -3.141593, 0.000000],accel_mss,speed_ms,0,blend_radius_m)
    |   movel(p[0.463662, -0.050600, -0.000100, 0.000000, -3.141593, 0.000000],accel_mss,speed_ms,0,blend_radius_m)
    |   movel(p[0.465046, -0.049389, -0.000100, 0.000000, -3.141593, 0.000000],accel_mss,speed_ms,0,blend_radius_m)
    |   movel(p[0.465674, -0.048815, -0.000100, 0.000000, -3.141593, 0.000000],accel_mss,speed_ms,0,blend_radius_m)
    |   movel(p[0.466024, -0.048462, -0.000100, 0.000000, -3.141593, 0.000000],accel_mss,speed_ms,0,0.000)
    |   movel(p[0.466100, -0.048284, -0.000100, 0.000000, -3.141593, 0.000000],accel_mss,speed_ms,0,0.000)
    |   movel(p[0.466175, -0.048109, -0.000100, 0.000000, -3.141593, 0.000000],accel_mss,speed_ms,0,0.000)
    |   movel(p[0.466251, -0.048011, -0.000100, 0.000000, -3.141593, 0.000000],accel_mss,speed_ms,0,0.000)
    |   movel(p[0.466339, -0.047926, -0.000100, 0.000000, -3.141593, 0.000000],accel_mss,speed_ms,0,0.000)
    |   movel(p[0.466466, -0.047728, -0.000100, 0.000000, -3.141593, 0.000000],accel_mss,speed_ms,0,0.000)
    |   movel(p[0.466476, -0.047461, -0.000100, 0.000000, -3.141593, 0.000000],accel_mss,speed_ms,0,0.000)
    |   movel(p[0.466366, -0.047153, -0.000100, 0.000000, -3.141593, 0.000000],accel_mss,speed_ms,0,0.000)
    |   movel(p[0.466145, -0.046841, -0.000100, 0.000000, 3.141593, 0.000000],accel_mss,speed_ms,0,0.000)
    |   movel(p[0.465548, -0.046565, -0.000100, 0.000000, -3.141593, 0.000000],accel_mss,speed_ms,0,blend_radius_m)
    |   movel(p[0.464410, -0.046659, -0.000100, 0.000000, -3.141593, 0.000000],accel_mss,speed_ms,0,blend_radius_m)
    |   movel(p[0.463226, -0.046995, -0.000100, 0.000000, -3.141593, 0.000000],accel_mss,speed_ms,0,blend_radius_m)
    |   movel(p[0.462406, -0.047517, -0.000100, 0.000000, -3.141593, 0.000000],accel_mss,speed_ms,0,blend_radius_m)
    |   movel(p[0.462219, -0.047714, -0.000100, 0.000000, -3.141593, 0.000000],accel_mss,speed_ms,0,0.000)
    |   movel(p[0.462054, -0.047931, -0.000100, 0.000000, -3.141593, 0.000000],accel_mss,speed_ms,0,0.000)
    |   movel(p[0.461930, -0.048136, -0.000100, 0.000000, 3.141593, 0.000000],accel_mss,speed_ms,0,0.000)
    |   movel(p[0.461881, -0.048288, -0.000100, 0.000000, -3.141593, 0.000000],accel_mss,speed_ms,0,0.000)
    |   movel(p[0.461796, -0.048554, -0.000100, 0.000000, -3.141593, 0.000000],accel_mss,speed_ms,0,0.000)
    |   movel(p[0.461670, -0.048579, -0.000100, 0.000000, -3.141593, 0.000000],accel_mss,speed_ms,0,0.000)
    |   movel(p[0.461539, -0.048366, -0.000100, 0.000000, 3.141593, 0.000000],accel_mss,speed_ms,0,0.000)
    |   movel(p[0.461461, -0.047928, -0.000100, 0.000000, -3.141593, 0.000000],accel_mss,speed_ms,0,0.000)
    |   movel(p[0.461423, -0.047591, -0.000100, 0.000000, -3.141593, 0.000000],accel_mss,speed_ms,0,0.000)
    |   movel(p[0.461386, -0.047253, -0.000100, 0.000000, -3.141593, 0.000000],accel_mss,speed_ms,0,0.000)
    |   movel(p[0.460916, -0.047208, -0.000100, 0.000000, 3.141593, 0.000000],accel_mss,speed_ms,0,0.000)
    |   movel(p[0.460446, -0.047163, -0.000100, 0.000000, 3.141593, 0.000000],accel_mss,speed_ms,0,0.000)
    |   movel(p[0.460079, -0.047122, -0.000100, 0.000000, 3.141593, 0.000000],accel_mss,speed_ms,0,0.000)
    |   movel(p[0.459753, -0.047071, -0.000100, 0.000000, 3.141593, 0.000000],accel_mss,speed_ms,0,0.000)
    |   movel(p[0.459485, -0.047017, -0.000100, 0.000000, 3.141593, 0.000000],accel_mss,speed_ms,0,0.000)
    |   movel(p[0.459354, -0.046967, -0.000100, 0.000000, -3.141593, 0.000000],accel_mss,speed_ms,0,0.000)
    |   movel(p[0.459201, -0.047147, -0.000100, 0.000000, 3.141593, 0.000000],accel_mss,speed_ms,0,0.000)
    |   movel(p[0.459124, -0.047305, -0.000100, 0.000000, 3.141593, 0.000000],accel_mss,speed_ms,0,0.000)
    |   movel(p[0.459023, -0.047492, -0.000100, 0.000000, -3.141593, 0.000000],accel_mss,speed_ms,0,0.000)
    |   movel(p[0.458890, -0.047643, -0.000100, 0.000000, -3.141593, 0.000000],accel_mss,speed_ms,0,0.000)
    |   movel(p[0.458733, -0.047751, -0.000100, 0.000000, -3.141593, 0.000000],accel_mss,speed_ms,0,0.000)
    |   movel(p[0.458560, -0.047811, -0.000100, 0.000000, 3.141593, 0.000000],accel_mss,speed_ms,0,0.000)
    |   movel(p[0.458354, -0.047834, -0.000100, 0.000000, -3.141593, 0.000000],accel_mss,speed_ms,0,0.000)
    |   movel(p[0.458239, -0.047800, -0.000100, 0.000000, -3.141593, 0.000000],accel_mss,speed_ms,0,0.000)
    |   movel(p[0.458171, -0.047702, -0.000100, 0.000000, -3.141593, 0.000000],accel_mss,speed_ms,0,0.000)
    |   movel(p[0.458131, -0.047502, -0.000100, 0.000000, -3.141593, 0.000000],accel_mss,speed_ms,0,0.000)
    |   movel(p[0.457902, -0.047103, -0.000100, 0.000000, -3.141593, 0.000000],accel_mss,speed_ms,0,0.000)
    |   movel(p[0.457185, -0.046645, -0.000100, 0.000000, -3.141593, 0.000000],accel_mss,speed_ms,0,blend_radius_m)
    |   movel(p[0.456135, -0.046169, -0.000100, 0.000000, -3.141593, 0.000000],accel_mss,speed_ms,0,blend_radius_m)
    |   movel(p[0.454770, -0.045708, -0.000100, 0.000000, 3.141593, 0.000000],accel_mss,speed_ms,0,blend_radius_m)
    |   movel(p[0.453282, -0.045277, -0.000100, 0.000000, -3.141593, 0.000000],accel_mss,speed_ms,0,blend_radius_m)
    |   movel(p[0.452301, -0.045042, -0.000100, 0.000000, -3.141593, 0.000000],accel_mss,speed_ms,0,blend_radius_m)
    |   movel(p[0.451428, -0.044908, -0.000100, 0.000000, 3.141593, 0.000000],accel_mss,speed_ms,0,blend_radius_m)
    |   movel(p[0.450358, -0.044819, -0.000100, 0.000000, -3.141593, 0.000000],accel_mss,speed_ms,0,blend_radius_m)
    |   movel(p[0.448589, -0.044869, -0.000100, 0.000000, -3.141593, 0.000000],accel_mss,speed_ms,0,blend_radius_m)
    |   movel(p[0.447046, -0.045232, -0.000100, 0.000000, 3.141593, 0.000000],accel_mss,speed_ms,0,blend_radius_m)
    |   movel(p[0.445650, -0.045936, -0.000100, 0.000000, -3.141593, 0.000000],accel_mss,speed_ms,0,blend_radius_m)
    |   movel(p[0.444323, -0.047009, -0.000100, 0.000000, -3.141593, 0.000000],accel_mss,speed_ms,0,blend_radius_m)
    |   movel(p[0.443936, -0.047400, -0.000100, 0.000000, -3.141593, 0.000000],accel_mss,speed_ms,0,blend_radius_m)
    |   movel(p[0.443608, -0.047756, -0.000100, 0.000000, -3.141593, 0.000000],accel_mss,speed_ms,0,0.000)
    |   movel(p[0.443349, -0.048063, -0.000100, 0.000000, -3.141593, 0.000000],accel_mss,speed_ms,0,0.000)
    |   movel(p[0.443311, -0.048168, -0.000100, 0.000000, -3.141593, 0.000000],accel_mss,speed_ms,0,0.000)
    |   movel(p[0.443246, -0.048345, -0.000100, 0.000000, -3.141593, 0.000000],accel_mss,speed_ms,0,0.000)
    |   movel(p[0.443174, -0.048442, -0.000100, 0.000000, -3.141593, 0.000000],accel_mss,speed_ms,0,0.000)
    |   movel(p[0.443089, -0.048525, -0.000100, 0.000000, -3.141593, 0.000000],accel_mss,speed_ms,0,0.000)
    |   movel(p[0.442785, -0.048892, -0.000100, 0.000000, -3.141593, 0.000000],accel_mss,speed_ms,0,0.000)
    |   movel(p[0.442450, -0.049569, -0.000100, 0.000000, -3.141593, 0.000000],accel_mss,speed_ms,0,blend_radius_m)
    |   movel(p[0.442185, -0.050264, -0.000100, 0.000000, -3.141593, 0.000000],accel_mss,speed_ms,0,blend_radius_m)
    |   movel(p[0.442183, -0.050619, -0.000100, 0.000000, -3.141593, 0.000000],accel_mss,speed_ms,0,0.000)
    |   movel(p[0.442180, -0.050845, -0.000100, 0.000000, 3.141593, 0.000000],accel_mss,speed_ms,0,0.000)
    |   movel(p[0.442046, -0.050917, -0.000100, 0.000000, 3.141593, 0.000000],accel_mss,speed_ms,0,0.000)
    |   movel(p[0.441755, -0.050767, -0.000100, 0.000000, -3.141593, 0.000000],accel_mss,speed_ms,0,0.000)
    |   movel(p[0.441361, -0.050403, -0.000100, 0.000000, -3.141593, 0.000000],accel_mss,speed_ms,0,blend_radius_m)
    |   movel(p[0.441154, -0.050202, -0.000100, 0.000000, -3.141593, 0.000000],accel_mss,speed_ms,0,0.000)
    |   movel(p[0.440952, -0.050033, -0.000100, 0.000000, -3.141593, 0.000000],accel_mss,speed_ms,0,0.000)
    |   movel(p[0.440776, -0.049907, -0.000100, 0.000000, -3.141593, 0.000000],accel_mss,speed_ms,0,0.000)
    |   movel(p[0.440595, -0.049855, -0.000100, 0.000000, -3.141593, 0.000000],accel_mss,speed_ms,0,0.000)
    |   movel(p[0.440456, -0.049764, -0.000100, 0.000000, -3.141593, 0.000000],accel_mss,speed_ms,0,0.000)
    |   movel(p[0.440301, -0.049638, -0.000100, 0.000000, -3.141593, 0.000000],accel_mss,speed_ms,0,0.000)
    |   movel(p[0.440150, -0.049490, -0.000100, 0.000000, -3.141593, 0.000000],accel_mss,speed_ms,0,0.000)
    |   movel(p[0.439273, -0.048753, -0.000100, 0.000000, -3.141593, 0.000000],accel_mss,speed_ms,0,blend_radius_m)
    |   movel(p[0.437959, -0.047989, -0.000100, 0.000000, -3.141593, 0.000000],accel_mss,speed_ms,0,blend_radius_m)
    |   movel(p[0.436512, -0.047340, -0.000100, 0.000000, -3.141593, 0.000000],accel_mss,speed_ms,0,blend_radius_m)
    |   movel(p[0.435201, -0.046951, -0.000100, 0.000000, 3.141593, 0.000000],accel_mss,speed_ms,0,blend_radius_m)
    |   movel(p[0.434266, -0.046804, -0.000100, 0.000000, -3.141593, 0.000000],accel_mss,speed_ms,0,blend_radius_m)
    |   movel(p[0.433264, -0.046741, -0.000100, 0.000000, -3.141593, 0.000000],accel_mss,speed_ms,0,blend_radius_m)
    |   movel(p[0.432226, -0.046764, -0.000100, 0.000000, -3.141593, 0.000000],accel_mss,speed_ms,0,blend_radius_m)
    |   movel(p[0.431181, -0.046872, -0.000100, 0.000000, -3.141593, 0.000000],accel_mss,speed_ms,0,blend_radius_m)
    |   movel(p[0.430489, -0.047022, -0.000100, 0.000000, -3.141593, 0.000000],accel_mss,speed_ms,0,blend_radius_m)
    |   movel(p[0.429759, -0.047278, -0.000100, 0.000000, 3.141593, 0.000000],accel_mss,speed_ms,0,blend_radius_m)
    |   movel(p[0.429005, -0.047634, -0.000100, 0.000000, -3.141593, 0.000000],accel_mss,speed_ms,0,blend_radius_m)
    |   movel(p[0.428236, -0.048085, -0.000100, 0.000000, -3.141593, 0.000000],accel_mss,speed_ms,0,blend_radius_m)
    |   movel(p[0.428047, -0.048204, -0.000100, 0.000000, -3.141593, 0.000000],accel_mss,speed_ms,0,0.000)
    |   movel(p[0.427852, -0.048320, -0.000100, 0.000000, -3.141593, 0.000000],accel_mss,speed_ms,0,0.000)
    |   movel(p[0.427677, -0.048419, -0.000100, 0.000000, -3.141593, 0.000000],accel_mss,speed_ms,0,0.000)
    |   movel(p[0.427561, -0.048477, -0.000100, 0.000000, -3.141593, 0.000000],accel_mss,speed_ms,0,0.000)
    |   movel(p[0.427440, -0.048542, -0.000100, 0.000000, -3.141593, 0.000000],accel_mss,speed_ms,0,0.000)
    |   movel(p[0.427241, -0.048673, -0.000100, 0.000000, -3.141593, 0.000000],accel_mss,speed_ms,0,0.000)
    |   movel(p[0.427015, -0.048833, -0.000100, 0.000000, -3.141593, 0.000000],accel_mss,speed_ms,0,0.000)
    |   movel(p[0.426789, -0.049003, -0.000100, 0.000000, -3.141593, 0.000000],accel_mss,speed_ms,0,0.000)
    |   movel(p[0.426570, -0.049166, -0.000100, 0.000000, -3.141593, 0.000000],accel_mss,speed_ms,0,0.000)
    |   movel(p[0.426362, -0.049303, -0.000100, 0.000000, -3.141593, 0.000000],accel_mss,speed_ms,0,0.000)
    |   movel(p[0.426185, -0.049407, -0.000100, 0.000000, -3.141593, 0.000000],accel_mss,speed_ms,0,0.000)
    |   movel(p[0.425895, -0.049508, -0.000100, 0.000000, -3.141593, 0.000000],accel_mss,speed_ms,0,0.000)
    |   movel(p[0.425633, -0.049787, -0.000100, 0.000000, -3.141593, 0.000000],accel_mss,speed_ms,0,0.000)
    |   movel(p[0.425426, -0.050098, -0.000100, 0.000000, -3.141593, 0.000000],accel_mss,speed_ms,0,0.000)
    |   movel(p[0.425430, -0.050278, -0.000100, 0.000000, 3.141593, 0.000000],accel_mss,speed_ms,0,0.000)
    |   movel(p[0.425518, -0.050358, -0.000100, 0.000000, -3.141593, 0.000000],accel_mss,speed_ms,0,0.000)
    |   movel(p[0.425769, -0.050474, -0.000100, 0.000000, -3.141593, 0.000000],accel_mss,speed_ms,0,0.000)
    |   movel(p[0.426084, -0.050594, -0.000100, 0.000000, -3.141593, 0.000000],accel_mss,speed_ms,0,0.000)
    |   movel(p[0.426436, -0.050705, -0.000100, 0.000000, -3.141593, 0.000000],accel_mss,speed_ms,0,0.000)
    |   movel(p[0.426791, -0.050813, -0.000100, 0.000000, 3.141593, 0.000000],accel_mss,speed_ms,0,0.000)
    |   movel(p[0.427113, -0.050925, -0.000100, 0.000000, -3.141593, 0.000000],accel_mss,speed_ms,0,0.000)
    |   movel(p[0.427378, -0.051030, -0.000100, 0.000000, -3.141593, 0.000000],accel_mss,speed_ms,0,0.000)
    |   movel(p[0.427478, -0.051095, -0.000100, 0.000000, -3.141593, 0.000000],accel_mss,speed_ms,0,0.000)
    |   movel(p[0.427652, -0.051189, -0.000100, 0.000000, -3.141593, 0.000000],accel_mss,speed_ms,0,0.000)
    |   movel(p[0.427763, -0.051219, -0.000100, 0.000000, -3.141593, 0.000000],accel_mss,speed_ms,0,0.000)
    |   movel(p[0.427868, -0.051228, -0.000100, 0.000000, -3.141593, 0.000000],accel_mss,speed_ms,0,0.000)
    |   movel(p[0.427996, -0.051245, -0.000100, 0.000000, -3.141593, 0.000000],accel_mss,speed_ms,0,0.000)
    |   movel(p[0.428191, -0.051302, -0.000100, 0.000000, -3.141593, 0.000000],accel_mss,speed_ms,0,0.000)
    |   movel(p[0.428408, -0.051384, -0.000100, 0.000000, -3.141593, 0.000000],accel_mss,speed_ms,0,0.000)
    |   movel(p[0.428619, -0.051480, -0.000100, 0.000000, 3.141593, 0.000000],accel_mss,speed_ms,0,0.000)
    |   movel(p[0.428871, -0.051578, -0.000100, 0.000000, -3.141593, 0.000000],accel_mss,speed_ms,0,0.000)
    |   movel(p[0.429196, -0.051656, -0.000100, 0.000000, -3.141593, 0.000000],accel_mss,speed_ms,0,0.000)
    |   movel(p[0.429546, -0.051705, -0.000100, 0.000000, 3.141593, 0.000000],accel_mss,speed_ms,0,0.000)
    |   movel(p[0.429880, -0.051718, -0.000100, 0.000000, 3.141593, 0.000000],accel_mss,speed_ms,0,0.000)
    |   movel(p[0.430348, -0.051709, -0.000100, 0.000000, 3.141593, 0.000000],accel_mss,speed_ms,0,0.000)
    |   movel(p[0.431407, -0.051688, -0.000100, 0.000000, -3.141593, 0.000000],accel_mss,speed_ms,0,blend_radius_m)
    |   movel(p[0.432666, -0.051663, -0.000100, 0.000000, -3.141593, 0.000000],accel_mss,speed_ms,0,blend_radius_m)
    |   movel(p[0.434016, -0.051637, -0.000100, 0.000000, -3.141593, 0.000000],accel_mss,speed_ms,0,blend_radius_m)
    |   movel(p[0.436330, -0.051628, -0.000100, 0.000000, -3.141593, 0.000000],accel_mss,speed_ms,0,blend_radius_m)
    |   movel(p[0.438154, -0.051710, -0.000100, 0.000000, -3.141593, 0.000000],accel_mss,speed_ms,0,blend_radius_m)
    |   movel(p[0.439648, -0.051889, -0.000100, 0.000000, -3.141593, 0.000000],accel_mss,speed_ms,0,blend_radius_m)
    |   movel(p[0.440930, -0.052177, -0.000100, 0.000000, -3.141593, 0.000000],accel_mss,speed_ms,0,blend_radius_m)
    |   movel(p[0.441461, -0.052399, -0.000100, 0.000000, -3.141593, 0.000000],accel_mss,speed_ms,0,blend_radius_m)
    |   movel(p[0.441439, -0.052551, -0.000100, 0.000000, -3.141593, 0.000000],accel_mss,speed_ms,0,0.000)
    |   movel(p[0.440742, -0.052636, -0.000100, 0.000000, 3.141593, 0.000000],accel_mss,speed_ms,0,blend_radius_m)
    |   movel(p[0.438884, -0.052649, -0.000100, 0.000000, -3.141593, 0.000000],accel_mss,speed_ms,0,blend_radius_m)
    |   movel(p[0.436472, -0.052692, -0.000100, 0.000000, -3.141593, 0.000000],accel_mss,speed_ms,0,blend_radius_m)
    |   movel(p[0.434674, -0.052841, -0.000100, 0.000000, -3.141593, 0.000000],accel_mss,speed_ms,0,blend_radius_m)
    |   movel(p[0.433000, -0.053144, -0.000100, 0.000000, 3.141593, 0.000000],accel_mss,speed_ms,0,blend_radius_m)
    |   movel(p[0.431011, -0.053668, -0.000100, 0.000000, -3.141593, 0.000000],accel_mss,speed_ms,0,blend_radius_m)
    |   movel(p[0.430081, -0.054014, -0.000100, 0.000000, -3.141593, 0.000000],accel_mss,speed_ms,0,blend_radius_m)
    |   movel(p[0.428740, -0.054657, -0.000100, 0.000000, -3.141593, 0.000000],accel_mss,speed_ms,0,blend_radius_m)
    |   movel(p[0.427448, -0.055345, -0.000100, 0.000000, 3.141593, 0.000000],accel_mss,speed_ms,0,blend_radius_m)
    |   movel(p[0.426825, -0.055791, -0.000100, 0.000000, -3.141593, 0.000000],accel_mss,speed_ms,0,blend_radius_m)
    |   movel(p[0.426714, -0.055882, -0.000100, 0.000000, 3.141593, 0.000000],accel_mss,speed_ms,0,0.000)
    |   movel(p[0.426599, -0.055959, -0.000100, 0.000000, -3.141593, 0.000000],accel_mss,speed_ms,0,0.000)
    |   movel(p[0.426496, -0.056013, -0.000100, 0.000000, -3.141593, 0.000000],accel_mss,speed_ms,0,0.000)
    |   movel(p[0.426194, -0.056124, -0.000100, 0.000000, -3.141593, 0.000000],accel_mss,speed_ms,0,0.000)
    |   movel(p[0.424446, -0.057871, -0.000100, 0.000000, -3.141593, 0.000000],accel_mss,speed_ms,0,blend_radius_m)
    |   movel(p[0.422707, -0.059625, -0.000100, 0.000000, -3.141593, 0.000000],accel_mss,speed_ms,0,blend_radius_m)
    |   movel(p[0.422611, -0.059858, -0.000100, 0.000000, -3.141593, 0.000000],accel_mss,speed_ms,0,0.000)
    |   movel(p[0.422435, -0.060143, -0.000100, 0.000000, -3.141593, 0.000000],accel_mss,speed_ms,0,0.000)
    |   movel(p[0.422241, -0.060367, -0.000100, 0.000000, 3.141593, 0.000000],accel_mss,speed_ms,0,0.000)
    |   movel(p[0.422011, -0.060603, -0.000100, 0.000000, -3.141593, 0.000000],accel_mss,speed_ms,0,0.000)
    |   movel(p[0.421781, -0.060840, -0.000100, 0.000000, 3.141593, 0.000000],accel_mss,speed_ms,0,0.000)
    |   movel(p[0.421587, -0.061065, -0.000100, 0.000000, -3.141593, 0.000000],accel_mss,speed_ms,0,0.000)
    |   movel(p[0.421441, -0.061259, -0.000100, 0.000000, -3.141593, 0.000000],accel_mss,speed_ms,0,0.000)
    |   movel(p[0.421378, -0.061448, -0.000100, 0.000000, -3.141593, 0.000000],accel_mss,speed_ms,0,0.000)
    |   movel(p[0.421191, -0.061684, -0.000100, 0.000000, -3.141593, 0.000000],accel_mss,speed_ms,0,0.000)
    |   movel(p[0.420948, -0.061959, -0.000100, 0.000000, -3.141593, 0.000000],accel_mss,speed_ms,0,0.000)
    |   movel(p[0.420661, -0.062253, -0.000100, 0.000000, 3.141593, 0.000000],accel_mss,speed_ms,0,0.000)
    |   movel(p[0.420374, -0.062545, -0.000100, 0.000000, -3.141593, 0.000000],accel_mss,speed_ms,0,0.000)
    |   movel(p[0.420131, -0.062810, -0.000100, 0.000000, -3.141593, 0.000000],accel_mss,speed_ms,0,0.000)
    |   movel(p[0.419937, -0.063037, -0.000100, 0.000000, -3.141593, 0.000000],accel_mss,speed_ms,0,0.000)
    |   movel(p[0.419938, -0.063156, -0.000100, 0.000000, -3.141593, 0.000000],accel_mss,speed_ms,0,0.000)
    |   movel(p[0.420032, -0.063194, -0.000100, 0.000000, -3.141593, 0.000000],accel_mss,speed_ms,0,0.000)
    |   movel(p[0.420165, -0.063220, -0.000100, 0.000000, -3.141593, 0.000000],accel_mss,speed_ms,0,0.000)
    |   movel(p[0.420323, -0.063229, -0.000100, 0.000000, -3.141593, 0.000000],accel_mss,speed_ms,0,0.000)
    |   movel(p[0.420947, -0.063187, -0.000100, 0.000000, -3.141593, 0.000000],accel_mss,speed_ms,0,blend_radius_m)
    |   movel(p[0.422817, -0.062921, -0.000100, 0.000000, -3.141593, 0.000000],accel_mss,speed_ms,0,blend_radius_m)
    |   movel(p[0.424652, -0.062642, -0.000100, 0.000000, -3.141593, 0.000000],accel_mss,speed_ms,0,blend_radius_m)
    |   movel(p[0.425461, -0.062476, -0.000100, 0.000000, 3.141593, 0.000000],accel_mss,speed_ms,0,blend_radius_m)
    |   movel(p[0.425762, -0.062409, -0.000100, 0.000000, -3.141593, 0.000000],accel_mss,speed_ms,0,0.000)
    |   movel(p[0.426313, -0.062308, -0.000100, 0.000000, -3.141593, 0.000000],accel_mss,speed_ms,0,blend_radius_m)
    |   movel(p[0.426959, -0.062197, -0.000100, 0.000000, 3.141593, 0.000000],accel_mss,speed_ms,0,blend_radius_m)
    |   movel(p[0.427625, -0.062091, -0.000100, 0.000000, -3.141593, 0.000000],accel_mss,speed_ms,0,blend_radius_m)
    |   movel(p[0.429897, -0.061671, -0.000100, 0.000000, -3.141593, 0.000000],accel_mss,speed_ms,0,blend_radius_m)
    |   movel(p[0.432170, -0.061106, -0.000100, 0.000000, -3.141593, 0.000000],accel_mss,speed_ms,0,blend_radius_m)
    |   movel(p[0.434165, -0.060482, -0.000100, 0.000000, -3.141593, 0.000000],accel_mss,speed_ms,0,blend_radius_m)
    |   movel(p[0.435511, -0.059884, -0.000100, 0.000000, -3.141593, 0.000000],accel_mss,speed_ms,0,blend_radius_m)
    |   movel(p[0.435849, -0.059698, -0.000100, 0.000000, -3.141593, 0.000000],accel_mss,speed_ms,0,0.000)
    |   movel(p[0.436182, -0.059516, -0.000100, 0.000000, -3.141593, 0.000000],accel_mss,speed_ms,0,0.000)
    |   movel(p[0.436469, -0.059359, -0.000100, 0.000000, -3.141593, 0.000000],accel_mss,speed_ms,0,0.000)
    |   movel(p[0.436636, -0.059268, -0.000100, 0.000000, 3.141593, 0.000000],accel_mss,speed_ms,0,0.000)
    |   movel(p[0.437115, -0.058929, -0.000100, 0.000000, -3.141593, 0.000000],accel_mss,speed_ms,0,blend_radius_m)
    |   movel(p[0.437893, -0.058196, -0.000100, 0.000000, -3.141593, 0.000000],accel_mss,speed_ms,0,blend_radius_m)
    |   movel(p[0.438646, -0.057417, -0.000100, 0.000000, -3.141593, 0.000000],accel_mss,speed_ms,0,blend_radius_m)
    |   movel(p[0.439085, -0.056853, -0.000100, 0.000000, 3.141593, 0.000000],accel_mss,speed_ms,0,blend_radius_m)
    |   movel(p[0.439445, -0.056301, -0.000100, 0.000000, -3.141593, 0.000000],accel_mss,speed_ms,0,blend_radius_m)
    |   movel(p[0.439681, -0.055922, -0.000100, 0.000000, -3.141593, 0.000000],accel_mss,speed_ms,0,0.000)
    |   movel(p[0.439851, -0.055626, -0.000100, 0.000000, -3.141593, 0.000000],accel_mss,speed_ms,0,0.000)
    |   movel(p[0.439990, -0.055353, -0.000100, 0.000000, -3.141593, 0.000000],accel_mss,speed_ms,0,0.000)
    |   movel(p[0.440078, -0.055205, -0.000100, 0.000000, -3.141593, 0.000000],accel_mss,speed_ms,0,0.000)
    |   movel(p[0.440242, -0.054996, -0.000100, 0.000000, -3.141593, 0.000000],accel_mss,speed_ms,0,0.000)
    |   movel(p[0.440440, -0.054771, -0.000100, 0.000000, -3.141593, 0.000000],accel_mss,speed_ms,0,0.000)
    |   movel(p[0.440648, -0.054559, -0.000100, 0.000000, -3.141593, 0.000000],accel_mss,speed_ms,0,0.000)
    |   movel(p[0.441075, -0.054235, -0.000100, 0.000000, -3.141593, 0.000000],accel_mss,speed_ms,0,blend_radius_m)
    |   movel(p[0.441328, -0.054272, -0.000100, 0.000000, -3.141593, 0.000000],accel_mss,speed_ms,0,0.000)
    |   movel(p[0.441480, -0.054613, -0.000100, 0.000000, -3.141593, 0.000000],accel_mss,speed_ms,0,0.000)
    |   movel(p[0.441531, -0.055516, -0.000100, 0.000000, -3.141593, 0.000000],accel_mss,speed_ms,0,blend_radius_m)
    |   movel(p[0.441432, -0.057098, -0.000100, 0.000000, 3.141593, 0.000000],accel_mss,speed_ms,0,blend_radius_m)
    |   movel(p[0.441054, -0.058447, -0.000100, 0.000000, -3.141593, 0.000000],accel_mss,speed_ms,0,blend_radius_m)
    |   movel(p[0.440335, -0.059723, -0.000100, 0.000000, -3.141593, 0.000000],accel_mss,speed_ms,0,blend_radius_m)
    |   movel(p[0.439195, -0.061091, -0.000100, 0.000000, -3.141593, 0.000000],accel_mss,speed_ms,0,blend_radius_m)
    |   movel(p[0.438896, -0.061393, -0.000100, 0.000000, 3.141593, 0.000000],accel_mss,speed_ms,0,0.000)
    |   movel(p[0.438617, -0.061647, -0.000100, 0.000000, -3.141593, 0.000000],accel_mss,speed_ms,0,0.000)
    |   movel(p[0.438378, -0.061844, -0.000100, 0.000000, -3.141593, 0.000000],accel_mss,speed_ms,0,0.000)
    |   movel(p[0.438280, -0.061878, -0.000100, 0.000000, -3.141593, 0.000000],accel_mss,speed_ms,0,0.000)
    |   movel(p[0.438061, -0.061986, -0.000100, 0.000000, 3.141593, 0.000000],accel_mss,speed_ms,0,0.000)
    |   movel(p[0.437913, -0.062105, -0.000100, 0.000000, -3.141593, 0.000000],accel_mss,speed_ms,0,0.000)
    |   movel(p[0.437769, -0.062245, -0.000100, 0.000000, 3.141593, 0.000000],accel_mss,speed_ms,0,0.000)
    |   movel(p[0.437603, -0.062403, -0.000100, 0.000000, -3.141593, 0.000000],accel_mss,speed_ms,0,0.000)
    |   movel(p[0.437388, -0.062574, -0.000100, 0.000000, -3.141593, 0.000000],accel_mss,speed_ms,0,0.000)
    |   movel(p[0.437160, -0.062732, -0.000100, 0.000000, -3.141593, 0.000000],accel_mss,speed_ms,0,0.000)
    |   movel(p[0.436955, -0.062849, -0.000100, 0.000000, -3.141593, 0.000000],accel_mss,speed_ms,0,0.000)
    |   movel(p[0.436759, -0.062950, -0.000100, 0.000000, 3.141593, 0.000000],accel_mss,speed_ms,0,0.000)
    |   movel(p[0.436558, -0.063056, -0.000100, 0.000000, 3.141593, 0.000000],accel_mss,speed_ms,0,0.000)
    |   movel(p[0.436379, -0.063153, -0.000100, 0.000000, -3.141593, 0.000000],accel_mss,speed_ms,0,0.000)
    |   movel(p[0.436261, -0.063221, -0.000100, 0.000000, 3.141593, 0.000000],accel_mss,speed_ms,0,0.000)
    |   movel(p[0.435731, -0.063509, -0.000100, 0.000000, -3.141593, 0.000000],accel_mss,speed_ms,0,blend_radius_m)
    |   movel(p[0.435148, -0.063773, -0.000100, 0.000000, 3.141593, 0.000000],accel_mss,speed_ms,0,blend_radius_m)
    |   movel(p[0.434608, -0.063977, -0.000100, 0.000000, -3.141593, 0.000000],accel_mss,speed_ms,0,blend_radius_m)
    |   movel(p[0.434240, -0.064058, -0.000100, 0.000000, -3.141593, 0.000000],accel_mss,speed_ms,0,0.000)
    |   movel(p[0.434005, -0.064093, -0.000100, 0.000000, -3.141593, 0.000000],accel_mss,speed_ms,0,0.000)
    |   movel(p[0.433649, -0.064161, -0.000100, 0.000000, -3.141593, 0.000000],accel_mss,speed_ms,0,0.000)
    |   movel(p[0.433252, -0.064246, -0.000100, 0.000000, -3.141593, 0.000000],accel_mss,speed_ms,0,0.000)
    |   movel(p[0.432866, -0.064337, -0.000100, 0.000000, -3.141593, 0.000000],accel_mss,speed_ms,0,0.000)
    |   movel(p[0.430657, -0.064762, -0.000100, 0.000000, -3.141593, 0.000000],accel_mss,speed_ms,0,blend_radius_m)
    |   movel(p[0.428237, -0.064985, -0.000100, 0.000000, -3.141593, 0.000000],accel_mss,speed_ms,0,blend_radius_m)
    |   movel(p[0.425735, -0.065001, -0.000100, 0.000000, -3.141593, 0.000000],accel_mss,speed_ms,0,blend_radius_m)
    |   movel(p[0.423280, -0.064805, -0.000100, 0.000000, -3.141593, 0.000000],accel_mss,speed_ms,0,blend_radius_m)
    |   movel(p[0.422495, -0.064719, -0.000100, 0.000000, -3.141593, 0.000000],accel_mss,speed_ms,0,blend_radius_m)
    |   movel(p[0.421618, -0.064646, -0.000100, 0.000000, -3.141593, 0.000000],accel_mss,speed_ms,0,blend_radius_m)
    |   movel(p[0.420784, -0.064596, -0.000100, 0.000000, -3.141593, 0.000000],accel_mss,speed_ms,0,blend_radius_m)
    |   movel(p[0.420142, -0.064580, -0.000100, 0.000000, -3.141593, 0.000000],accel_mss,speed_ms,0,blend_radius_m)
    |   movel(p[0.419266, -0.064590, -0.000100, 0.000000, -3.141593, 0.000000],accel_mss,speed_ms,0,blend_radius_m)
    |   movel(p[0.418898, -0.064647, -0.000100, 0.000000, -3.141593, 0.000000],accel_mss,speed_ms,0,0.000)
    |   movel(p[0.418620, -0.064789, -0.000100, 0.000000, 3.141593, 0.000000],accel_mss,speed_ms,0,0.000)
    |   movel(p[0.418243, -0.065121, -0.000100, 0.000000, 3.141593, 0.000000],accel_mss,speed_ms,0,blend_radius_m)
    |   movel(p[0.418019, -0.065321, -0.000100, 0.000000, -3.141593, 0.000000],accel_mss,speed_ms,0,0.000)
    |   movel(p[0.417804, -0.065474, -0.000100, 0.000000, -3.141593, 0.000000],accel_mss,speed_ms,0,0.000)
    |   movel(p[0.417622, -0.065570, -0.000100, 0.000000, -3.141593, 0.000000],accel_mss,speed_ms,0,0.000)
    |   movel(p[0.417386, -0.065301, -0.000100, 0.000000, -3.141593, 0.000000],accel_mss,speed_ms,0,0.000)
    |   movel(p[0.417445, -0.064205, -0.000100, 0.000000, -3.141593, 0.000000],accel_mss,speed_ms,0,blend_radius_m)
    |   movel(p[0.417580, -0.063025, -0.000100, 0.000000, -3.141593, 0.000000],accel_mss,speed_ms,0,blend_radius_m)
    |   movel(p[0.417799, -0.061986, -0.000100, 0.000000, -3.141593, 0.000000],accel_mss,speed_ms,0,blend_radius_m)
    |   movel(p[0.418133, -0.060819, -0.000100, 0.000000, -3.141593, 0.000000],accel_mss,speed_ms,0,blend_radius_m)
    |   movel(p[0.418418, -0.060032, -0.000100, 0.000000, -3.141593, 0.000000],accel_mss,speed_ms,0,blend_radius_m)
    |   movel(p[0.418772, -0.059306, -0.000100, 0.000000, -3.141593, 0.000000],accel_mss,speed_ms,0,blend_radius_m)
    |   movel(p[0.419331, -0.058353, -0.000100, 0.000000, -3.141593, 0.000000],accel_mss,speed_ms,0,blend_radius_m)
    |   movel(p[0.419444, -0.058165, -0.000100, 0.000000, -3.141593, 0.000000],accel_mss,speed_ms,0,0.000)
    |   movel(p[0.419555, -0.057969, -0.000100, 0.000000, -3.141593, 0.000000],accel_mss,speed_ms,0,0.000)
    |   movel(p[0.419650, -0.057794, -0.000100, 0.000000, -3.141593, 0.000000],accel_mss,speed_ms,0,0.000)
    |   movel(p[0.419706, -0.057678, -0.000100, 0.000000, -3.141593, 0.000000],accel_mss,speed_ms,0,0.000)
    |   movel(p[0.419931, -0.057332, -0.000100, 0.000000, -3.141593, 0.000000],accel_mss,speed_ms,0,0.000)
    |   movel(p[0.420584, -0.056650, -0.000100, 0.000000, -3.141593, 0.000000],accel_mss,speed_ms,0,blend_radius_m)
    |   movel(p[0.421281, -0.055964, -0.000100, 0.000000, -3.141593, 0.000000],accel_mss,speed_ms,0,blend_radius_m)
    |   movel(p[0.421495, -0.055878, -0.000100, 0.000000, -3.141593, 0.000000],accel_mss,speed_ms,0,0.000)
    |   movel(p[0.421694, -0.055790, -0.000100, 0.000000, -3.141593, 0.000000],accel_mss,speed_ms,0,0.000)
    |   movel(p[0.421820, -0.055693, -0.000100, 0.000000, -3.141593, 0.000000],accel_mss,speed_ms,0,0.000)
    |   movel(p[0.421936, -0.055578, -0.000100, 0.000000, -3.141593, 0.000000],accel_mss,speed_ms,0,0.000)
    |   movel(p[0.422053, -0.055464, -0.000100, 0.000000, 3.141593, 0.000000],accel_mss,speed_ms,0,0.000)
    |   movel(p[0.422180, -0.055366, -0.000100, 0.000000, -3.141593, 0.000000],accel_mss,speed_ms,0,0.000)
    |   movel(p[0.422299, -0.055298, -0.000100, 0.000000, -3.141593, 0.000000],accel_mss,speed_ms,0,0.000)
    |   movel(p[0.422472, -0.055259, -0.000100, 0.000000, -3.141593, 0.000000],accel_mss,speed_ms,0,0.000)
    |   movel(p[0.422589, -0.055193, -0.000100, 0.000000, -3.141593, 0.000000],accel_mss,speed_ms,0,0.000)
    |   movel(p[0.422713, -0.055100, -0.000100, 0.000000, -3.141593, 0.000000],accel_mss,speed_ms,0,0.000)
    |   movel(p[0.422826, -0.054989, -0.000100, 0.000000, -3.141593, 0.000000],accel_mss,speed_ms,0,0.000)
    |   movel(p[0.422960, -0.054861, -0.000100, 0.000000, -3.141593, 0.000000],accel_mss,speed_ms,0,0.000)
    |   movel(p[0.423151, -0.054713, -0.000100, 0.000000, -3.141593, 0.000000],accel_mss,speed_ms,0,0.000)
    |   movel(p[0.423361, -0.054570, -0.000100, 0.000000, -3.141593, 0.000000],accel_mss,speed_ms,0,0.000)
    |   movel(p[0.423562, -0.054456, -0.000100, 0.000000, -3.141593, 0.000000],accel_mss,speed_ms,0,0.000)
    |   movel(p[0.424635, -0.053890, -0.000100, 0.000000, -3.141593, 0.000000],accel_mss,speed_ms,0,blend_radius_m)
    |   movel(p[0.425553, -0.053376, -0.000100, 0.000000, -3.141593, 0.000000],accel_mss,speed_ms,0,blend_radius_m)
    |   movel(p[0.426333, -0.052919, -0.000100, 0.000000, -3.141593, 0.000000],accel_mss,speed_ms,0,blend_radius_m)
    |   movel(p[0.426413, -0.052805, -0.000100, 0.000000, -3.141593, 0.000000],accel_mss,speed_ms,0,0.000)
    |   movel(p[0.426247, -0.052500, -0.000100, 0.000000, -3.141593, 0.000000],accel_mss,speed_ms,0,0.000)
    |   movel(p[0.425151, -0.052094, -0.000100, 0.000000, -3.141593, 0.000000],accel_mss,speed_ms,0,blend_radius_m)
    |   movel(p[0.423717, -0.051698, -0.000100, 0.000000, -3.141593, 0.000000],accel_mss,speed_ms,0,blend_radius_m)
    |   movel(p[0.422038, -0.051374, -0.000100, 0.000000, -3.141593, 0.000000],accel_mss,speed_ms,0,blend_radius_m)
    |   movel(p[0.421559, -0.051284, -0.000100, 0.000000, 3.141593, 0.000000],accel_mss,speed_ms,0,0.000)
    |   movel(p[0.421200, -0.051185, -0.000100, 0.000000, 3.141593, 0.000000],accel_mss,speed_ms,0,0.000)
    |   movel(p[0.420951, -0.051081, -0.000100, 0.000000, -3.141593, 0.000000],accel_mss,speed_ms,0,0.000)
    |   movel(p[0.420854, -0.050973, -0.000100, 0.000000, -3.141593, 0.000000],accel_mss,speed_ms,0,0.000)
    |   movel(p[0.420844, -0.050842, -0.000100, 0.000000, -3.141593, 0.000000],accel_mss,speed_ms,0,0.000)
    |   movel(p[0.420912, -0.050594, -0.000100, 0.000000, -3.141593, 0.000000],accel_mss,speed_ms,0,0.000)
    |   movel(p[0.421024, -0.050302, -0.000100, 0.000000, -3.141593, 0.000000],accel_mss,speed_ms,0,0.000)
    |   movel(p[0.421173, -0.049998, -0.000100, 0.000000, -3.141593, 0.000000],accel_mss,speed_ms,0,0.000)
    |   movel(p[0.421323, -0.049704, -0.000100, 0.000000, -3.141593, 0.000000],accel_mss,speed_ms,0,0.000)
    |   movel(p[0.421437, -0.049445, -0.000100, 0.000000, -3.141593, 0.000000],accel_mss,speed_ms,0,0.000)
    |   movel(p[0.421516, -0.049230, -0.000100, 0.000000, -3.141593, 0.000000],accel_mss,speed_ms,0,0.000)
    |   movel(p[0.421358, -0.049126, -0.000100, 0.000000, -3.141593, 0.000000],accel_mss,speed_ms,0,0.000)
    |   movel(p[0.421154, -0.049208, -0.000100, 0.000000, -3.141593, 0.000000],accel_mss,speed_ms,0,0.000)
    |   movel(p[0.420948, -0.049384, -0.000100, 0.000000, -3.141593, 0.000000],accel_mss,speed_ms,0,0.000)
    |   movel(p[0.420802, -0.049612, -0.000100, 0.000000, -3.141593, 0.000000],accel_mss,speed_ms,0,0.000)
    |   movel(p[0.420615, -0.049996, -0.000100, 0.000000, -3.141593, 0.000000],accel_mss,speed_ms,0,0.000)
    |   movel(p[0.420417, -0.050345, -0.000100, 0.000000, -3.141593, 0.000000],accel_mss,speed_ms,0,0.000)
    |   movel(p[0.420213, -0.050651, -0.000100, 0.000000, -3.141593, 0.000000],accel_mss,speed_ms,0,0.000)
    |   movel(p[0.420010, -0.050902, -0.000100, 0.000000, -3.141593, 0.000000],accel_mss,speed_ms,0,0.000)
    |   movel(p[0.419915, -0.051016, -0.000100, 0.000000, -3.141593, 0.000000],accel_mss,speed_ms,0,0.000)
    |   movel(p[0.419834, -0.051133, -0.000100, 0.000000, 3.141593, 0.000000],accel_mss,speed_ms,0,0.000)
    |   movel(p[0.419776, -0.051236, -0.000100, 0.000000, -3.141593, 0.000000],accel_mss,speed_ms,0,0.000)
    |   movel(p[0.419742, -0.051374, -0.000100, 0.000000, -3.141593, 0.000000],accel_mss,speed_ms,0,0.000)
    |   movel(p[0.419651, -0.051533, -0.000100, 0.000000, -3.141593, 0.000000],accel_mss,speed_ms,0,0.000)
    |   movel(p[0.419530, -0.051719, -0.000100, 0.000000, -3.141593, 0.000000],accel_mss,speed_ms,0,0.000)
    |   movel(p[0.419386, -0.051917, -0.000100, 0.000000, -3.141593, 0.000000],accel_mss,speed_ms,0,0.000)
    |   movel(p[0.419242, -0.052115, -0.000100, 0.000000, -3.141593, 0.000000],accel_mss,speed_ms,0,0.000)
    |   movel(p[0.419121, -0.052306, -0.000100, 0.000000, -3.141593, 0.000000],accel_mss,speed_ms,0,0.000)
    |   movel(p[0.419031, -0.052469, -0.000100, 0.000000, 3.141593, 0.000000],accel_mss,speed_ms,0,0.000)
    |   movel(p[0.418996, -0.052616, -0.000100, 0.000000, -3.141593, 0.000000],accel_mss,speed_ms,0,0.000)
    |   movel(p[0.418881, -0.052789, -0.000100, 0.000000, -3.141593, 0.000000],accel_mss,speed_ms,0,0.000)
    |   movel(p[0.418801, -0.052866, -0.000100, 0.000000, -3.141593, 0.000000],accel_mss,speed_ms,0,0.000)
    |   movel(p[0.418713, -0.052961, -0.000100, 0.000000, -3.141593, 0.000000],accel_mss,speed_ms,0,0.000)
    |   movel(p[0.418623, -0.053104, -0.000100, 0.000000, -3.141593, 0.000000],accel_mss,speed_ms,0,0.000)
    |   movel(p[0.418546, -0.053268, -0.000100, 0.000000, -3.141593, 0.000000],accel_mss,speed_ms,0,0.000)
    |   movel(p[0.418493, -0.053430, -0.000100, 0.000000, -3.141593, 0.000000],accel_mss,speed_ms,0,0.000)
    |   movel(p[0.418430, -0.053613, -0.000100, 0.000000, -3.141593, 0.000000],accel_mss,speed_ms,0,0.000)
    |   movel(p[0.418316, -0.053846, -0.000100, 0.000000, -3.141593, 0.000000],accel_mss,speed_ms,0,0.000)
    |   movel(p[0.418176, -0.054088, -0.000100, 0.000000, -3.141593, 0.000000],accel_mss,speed_ms,0,0.000)
    |   movel(p[0.418028, -0.054301, -0.000100, 0.000000, -3.141593, 0.000000],accel_mss,speed_ms,0,0.000)
    |   movel(p[0.417887, -0.054492, -0.000100, 0.000000, -3.141593, 0.000000],accel_mss,speed_ms,0,0.000)
    |   movel(p[0.417769, -0.054668, -0.000100, 0.000000, -3.141593, 0.000000],accel_mss,speed_ms,0,0.000)
    |   movel(p[0.417677, -0.054819, -0.000100, 0.000000, 3.141593, 0.000000],accel_mss,speed_ms,0,0.000)
    |   movel(p[0.417647, -0.054947, -0.000100, 0.000000, -3.141593, 0.000000],accel_mss,speed_ms,0,0.000)
    |   movel(p[0.417459, -0.055375, -0.000100, 0.000000, -3.141593, 0.000000],accel_mss,speed_ms,0,0.000)
    |   movel(p[0.417237, -0.055870, -0.000100, 0.000000, -3.141593, 0.000000],accel_mss,speed_ms,0,blend_radius_m)
    |   movel(p[0.416974, -0.056438, -0.000100, 0.000000, -3.141593, 0.000000],accel_mss,speed_ms,0,blend_radius_m)
    |   movel(p[0.416701, -0.057024, -0.000100, 0.000000, -3.141593, 0.000000],accel_mss,speed_ms,0,blend_radius_m)
    |   movel(p[0.416448, -0.057572, -0.000100, 0.000000, -3.141593, 0.000000],accel_mss,speed_ms,0,blend_radius_m)
    |   movel(p[0.416238, -0.058034, -0.000100, 0.000000, -3.141593, 0.000000],accel_mss,speed_ms,0,blend_radius_m)
    |   movel(p[0.416149, -0.058241, -0.000100, 0.000000, 3.141593, 0.000000],accel_mss,speed_ms,0,0.000)
    |   movel(p[0.416086, -0.058394, -0.000100, 0.000000, -3.141593, 0.000000],accel_mss,speed_ms,0,0.000)
    |   movel(p[0.416009, -0.058578, -0.000100, 0.000000, -3.141593, 0.000000],accel_mss,speed_ms,0,0.000)
    |   movel(p[0.415931, -0.058762, -0.000100, 0.000000, 3.141593, 0.000000],accel_mss,speed_ms,0,0.000)
    |   movel(p[0.415865, -0.058916, -0.000100, 0.000000, 3.141593, 0.000000],accel_mss,speed_ms,0,0.000)
    |   movel(p[0.415789, -0.059100, -0.000100, 0.000000, -3.141593, 0.000000],accel_mss,speed_ms,0,0.000)
    |   movel(p[0.415669, -0.059408, -0.000100, 0.000000, -3.141593, 0.000000],accel_mss,speed_ms,0,0.000)
    |   movel(p[0.415535, -0.059761, -0.000100, 0.000000, -3.141593, 0.000000],accel_mss,speed_ms,0,0.000)
    |   movel(p[0.415404, -0.060116, -0.000100, 0.000000, -3.141593, 0.000000],accel_mss,speed_ms,0,0.000)
    |   movel(p[0.415275, -0.060446, -0.000100, 0.000000, -3.141593, 0.000000],accel_mss,speed_ms,0,0.000)
    |   movel(p[0.415148, -0.060725, -0.000100, 0.000000, -3.141593, 0.000000],accel_mss,speed_ms,0,0.000)
    |   movel(p[0.415033, -0.060944, -0.000100, 0.000000, -3.141593, 0.000000],accel_mss,speed_ms,0,0.000)
    |   movel(p[0.414921, -0.060957, -0.000100, 0.000000, -3.141593, 0.000000],accel_mss,speed_ms,0,0.000)
    |   movel(p[0.414846, -0.060879, -0.000100, 0.000000, -3.141593, 0.000000],accel_mss,speed_ms,0,0.000)
    |   movel(p[0.414767, -0.060770, -0.000100, 0.000000, 3.141593, 0.000000],accel_mss,speed_ms,0,0.000)
    |   movel(p[0.414695, -0.060641, -0.000100, 0.000000, -3.141593, 0.000000],accel_mss,speed_ms,0,0.000)
    |   movel(p[0.414388, -0.059986, -0.000100, 0.000000, 3.141593, 0.000000],accel_mss,speed_ms,0,blend_radius_m)
    |   movel(p[0.414060, -0.059220, -0.000100, 0.000000, -3.141593, 0.000000],accel_mss,speed_ms,0,blend_radius_m)
    |   movel(p[0.413760, -0.058461, -0.000100, 0.000000, -3.141593, 0.000000],accel_mss,speed_ms,0,blend_radius_m)
    |   movel(p[0.413536, -0.057828, -0.000100, 0.000000, -3.141593, 0.000000],accel_mss,speed_ms,0,blend_radius_m)
    |   movel(p[0.413419, -0.057491, -0.000100, 0.000000, 3.141593, 0.000000],accel_mss,speed_ms,0,0.000)
    |   movel(p[0.413287, -0.057159, -0.000100, 0.000000, -3.141593, 0.000000],accel_mss,speed_ms,0,0.000)
    |   movel(p[0.413160, -0.056874, -0.000100, 0.000000, -3.141593, 0.000000],accel_mss,speed_ms,0,0.000)
    |   movel(p[0.413064, -0.056707, -0.000100, 0.000000, -3.141593, 0.000000],accel_mss,speed_ms,0,0.000)
    |   movel(p[0.412986, -0.056576, -0.000100, 0.000000, -3.141593, 0.000000],accel_mss,speed_ms,0,0.000)
    |   movel(p[0.412921, -0.056426, -0.000100, 0.000000, -3.141593, 0.000000],accel_mss,speed_ms,0,0.000)
    |   movel(p[0.412875, -0.056281, -0.000100, 0.000000, -3.141593, 0.000000],accel_mss,speed_ms,0,0.000)
    |   movel(p[0.412861, -0.056165, -0.000100, 0.000000, 3.141593, 0.000000],accel_mss,speed_ms,0,0.000)
    |   movel(p[0.412838, -0.056007, -0.000100, 0.000000, -3.141593, 0.000000],accel_mss,speed_ms,0,0.000)
    |   movel(p[0.412706, -0.055578, -0.000100, 0.000000, 3.141593, 0.000000],accel_mss,speed_ms,0,0.000)
    |   movel(p[0.412536, -0.055068, -0.000100, 0.000000, -3.141593, 0.000000],accel_mss,speed_ms,0,blend_radius_m)
    |   movel(p[0.412334, -0.054511, -0.000100, 0.000000, -3.141593, 0.000000],accel_mss,speed_ms,0,blend_radius_m)
    |   movel(p[0.412127, -0.053939, -0.000100, 0.000000, -3.141593, 0.000000],accel_mss,speed_ms,0,blend_radius_m)
    |   movel(p[0.411939, -0.053385, -0.000100, 0.000000, 3.141593, 0.000000],accel_mss,speed_ms,0,blend_radius_m)
    |   movel(p[0.411789, -0.052910, -0.000100, 0.000000, -3.141593, 0.000000],accel_mss,speed_ms,0,0.000)
    |   movel(p[0.411727, -0.052653, -0.000100, 0.000000, -3.141593, 0.000000],accel_mss,speed_ms,0,0.000)
    |   movel(p[0.411673, -0.052407, -0.000100, 0.000000, -3.141593, 0.000000],accel_mss,speed_ms,0,0.000)
    |   movel(p[0.411561, -0.051988, -0.000100, 0.000000, -3.141593, 0.000000],accel_mss,speed_ms,0,0.000)
    |   movel(p[0.411423, -0.051507, -0.000100, 0.000000, -3.141593, 0.000000],accel_mss,speed_ms,0,blend_radius_m)
    |   movel(p[0.411275, -0.051021, -0.000100, 0.000000, -3.141593, 0.000000],accel_mss,speed_ms,0,blend_radius_m)
    |   movel(p[0.411021, -0.050177, -0.000100, 0.000000, -3.141593, 0.000000],accel_mss,speed_ms,0,blend_radius_m)
    |   movel(p[0.410804, -0.049379, -0.000100, 0.000000, 3.141593, 0.000000],accel_mss,speed_ms,0,blend_radius_m)
    |   movel(p[0.410638, -0.048681, -0.000100, 0.000000, -3.141593, 0.000000],accel_mss,speed_ms,0,blend_radius_m)
    |   movel(p[0.410541, -0.048153, -0.000100, 0.000000, -3.141593, 0.000000],accel_mss,speed_ms,0,blend_radius_m)
    |   movel(p[0.410510, -0.047961, -0.000100, 0.000000, -3.141593, 0.000000],accel_mss,speed_ms,0,0.000)
    |   movel(p[0.410419, -0.047471, -0.000100, 0.000000, -3.141593, 0.000000],accel_mss,speed_ms,0,0.000)
    |   movel(p[0.410307, -0.046887, -0.000100, 0.000000, -3.141593, 0.000000],accel_mss,speed_ms,0,blend_radius_m)
    |   movel(p[0.410183, -0.046252, -0.000100, 0.000000, -3.141593, 0.000000],accel_mss,speed_ms,0,blend_radius_m)
    |   movel(p[0.409602, -0.042512, -0.000100, 0.000000, -3.141593, 0.000000],accel_mss,speed_ms,0,blend_radius_m)
    |   movel(p[0.409435, -0.039255, -0.000100, 0.000000, 3.141593, 0.000000],accel_mss,speed_ms,0,blend_radius_m)
    |   movel(p[0.409674, -0.036397, -0.000100, 0.000000, 3.141593, 0.000000],accel_mss,speed_ms,0,blend_radius_m)
    |   movel(p[0.410323, -0.033866, -0.000100, 0.000000, -3.141593, 0.000000],accel_mss,speed_ms,0,blend_radius_m)
    |   movel(p[0.410426, -0.033564, -0.000100, 0.000000, -3.141593, 0.000000],accel_mss,speed_ms,0,0.000)
    |   movel(p[0.410499, -0.033310, -0.000100, 0.000000, -3.141593, 0.000000],accel_mss,speed_ms,0,0.000)
    |   movel(p[0.410547, -0.033107, -0.000100, 0.000000, 3.141593, 0.000000],accel_mss,speed_ms,0,0.000)
    |   movel(p[0.410548, -0.032957, -0.000100, 0.000000, -3.141593, 0.000000],accel_mss,speed_ms,0,0.000)
    |   movel(p[0.410621, -0.032824, -0.000100, 0.000000, -3.141593, 0.000000],accel_mss,speed_ms,0,0.000)
    |   movel(p[0.410724, -0.032666, -0.000100, 0.000000, -3.141593, 0.000000],accel_mss,speed_ms,0,0.000)
    |   movel(p[0.410861, -0.032448, -0.000100, 0.000000, -3.141593, 0.000000],accel_mss,speed_ms,0,0.000)
    |   movel(p[0.411049, -0.032112, -0.000100, 0.000000, 3.141593, 0.000000],accel_mss,speed_ms,0,0.000)
    |   movel(p[0.411250, -0.031732, -0.000100, 0.000000, -3.141593, 0.000000],accel_mss,speed_ms,0,0.000)
    |   movel(p[0.411435, -0.031359, -0.000100, 0.000000, -3.141593, 0.000000],accel_mss,speed_ms,0,0.000)
    |   movel(p[0.411737, -0.030836, -0.000100, 0.000000, 3.141593, 0.000000],accel_mss,speed_ms,0,blend_radius_m)
    |   movel(p[0.412168, -0.030264, -0.000100, 0.000000, 3.141593, 0.000000],accel_mss,speed_ms,0,blend_radius_m)
    |   movel(p[0.412782, -0.029572, -0.000100, 0.000000, 3.141593, 0.000000],accel_mss,speed_ms,0,blend_radius_m)
    |   movel(p[0.413675, -0.028655, -0.000100, 0.000000, 3.141593, 0.000000],accel_mss,speed_ms,0,blend_radius_m)
    |   movel(p[0.414751, -0.027598, -0.000100, 0.000000, -3.141593, 0.000000],accel_mss,speed_ms,0,blend_radius_m)
    |   movel(p[0.415338, -0.027091, -0.000100, 0.000000, -3.141593, 0.000000],accel_mss,speed_ms,0,blend_radius_m)
    |   movel(p[0.415816, -0.026793, -0.000100, 0.000000, -3.141593, 0.000000],accel_mss,speed_ms,0,blend_radius_m)
    |   movel(p[0.416379, -0.026569, -0.000100, 0.000000, -3.141593, 0.000000],accel_mss,speed_ms,0,blend_radius_m)
    |   movel(p[0.417180, -0.026376, -0.000100, 0.000000, -3.141593, 0.000000],accel_mss,speed_ms,0,blend_radius_m)
    |   movel(p[0.417929, -0.026307, -0.000100, 0.000000, -3.141593, 0.000000],accel_mss,speed_ms,0,blend_radius_m)
    |   movel(p[0.418673, -0.026361, -0.000100, 0.000000, -3.141593, 0.000000],accel_mss,speed_ms,0,blend_radius_m)
    |   movel(p[0.419454, -0.026537, -0.000100, 0.000000, 3.141593, 0.000000],accel_mss,speed_ms,0,blend_radius_m)
    |   movel(p[0.420112, -0.026801, -0.000100, 0.000000, -3.141593, 0.000000],accel_mss,speed_ms,0,blend_radius_m)
    |   movel(p[0.420649, -0.027165, -0.000100, 0.000000, 3.141593, 0.000000],accel_mss,speed_ms,0,blend_radius_m)
    |   movel(p[0.421087, -0.027650, -0.000100, 0.000000, -3.141593, 0.000000],accel_mss,speed_ms,0,blend_radius_m)
    |   movel(p[0.421452, -0.028278, -0.000100, 0.000000, -3.141593, 0.000000],accel_mss,speed_ms,0,blend_radius_m)
    |   movel(p[0.421648, -0.028745, -0.000100, 0.000000, 3.141593, 0.000000],accel_mss,speed_ms,0,blend_radius_m)
    |   movel(p[0.421792, -0.029191, -0.000100, 0.000000, 3.141593, 0.000000],accel_mss,speed_ms,0,0.000)
    |   movel(p[0.421874, -0.029556, -0.000100, 0.000000, 3.141593, 0.000000],accel_mss,speed_ms,0,0.000)
    |   movel(p[0.421776, -0.029620, -0.000100, 0.000000, -3.141593, 0.000000],accel_mss,speed_ms,0,0.000)
    |   movel(p[0.421636, -0.029560, -0.000100, 0.000000, -3.141593, 0.000000],accel_mss,speed_ms,0,0.000)
    |   movel(p[0.421472, -0.029484, -0.000100, 0.000000, 3.141593, 0.000000],accel_mss,speed_ms,0,0.000)
    |   movel(p[0.421289, -0.029395, -0.000100, 0.000000, -3.141593, 0.000000],accel_mss,speed_ms,0,0.000)
    |   movel(p[0.420668, -0.029184, -0.000100, 0.000000, -3.141593, 0.000000],accel_mss,speed_ms,0,blend_radius_m)
    |   movel(p[0.419744, -0.029051, -0.000100, 0.000000, -3.141593, 0.000000],accel_mss,speed_ms,0,blend_radius_m)
    |   movel(p[0.418804, -0.029009, -0.000100, 0.000000, 3.141593, 0.000000],accel_mss,speed_ms,0,blend_radius_m)
    |   movel(p[0.418120, -0.029096, -0.000100, 0.000000, -3.141593, 0.000000],accel_mss,speed_ms,0,blend_radius_m)
    |   movel(p[0.417453, -0.029381, -0.000100, 0.000000, -3.141593, 0.000000],accel_mss,speed_ms,0,blend_radius_m)
    |   movel(p[0.416864, -0.029868, -0.000100, 0.000000, 3.141593, 0.000000],accel_mss,speed_ms,0,blend_radius_m)
    |   movel(p[0.416415, -0.030502, -0.000100, 0.000000, -3.141593, 0.000000],accel_mss,speed_ms,0,blend_radius_m)
    |   movel(p[0.416158, -0.031216, -0.000100, 0.000000, -3.141593, 0.000000],accel_mss,speed_ms,0,blend_radius_m)
    |   movel(p[0.416026, -0.032451, -0.000100, 0.000000, -3.141593, 0.000000],accel_mss,speed_ms,0,blend_radius_m)
    |   movel(p[0.416117, -0.033794, -0.000100, 0.000000, -3.141593, 0.000000],accel_mss,speed_ms,0,blend_radius_m)
    |   movel(p[0.416416, -0.035122, -0.000100, 0.000000, -3.141593, 0.000000],accel_mss,speed_ms,0,blend_radius_m)
    |   movel(p[0.416903, -0.036313, -0.000100, 0.000000, -3.141593, 0.000000],accel_mss,speed_ms,0,blend_radius_m)
    |   movel(p[0.417313, -0.037037, -0.000100, 0.000000, -3.141593, 0.000000],accel_mss,speed_ms,0,blend_radius_m)
    |   movel(p[0.417655, -0.037474, -0.000100, 0.000000, -3.141593, 0.000000],accel_mss,speed_ms,0,blend_radius_m)
    |   movel(p[0.418069, -0.037800, -0.000100, 0.000000, -3.141593, 0.000000],accel_mss,speed_ms,0,blend_radius_m)
    |   movel(p[0.418706, -0.038141, -0.000100, 0.000000, -3.141593, 0.000000],accel_mss,speed_ms,0,blend_radius_m)
    |   movel(p[0.419665, -0.038458, -0.000100, 0.000000, -3.141593, 0.000000],accel_mss,speed_ms,0,blend_radius_m)
    |   movel(p[0.420744, -0.038564, -0.000100, 0.000000, 3.141593, 0.000000],accel_mss,speed_ms,0,blend_radius_m)
    |   movel(p[0.421818, -0.038457, -0.000100, 0.000000, 3.141593, 0.000000],accel_mss,speed_ms,0,blend_radius_m)
    |   movel(p[0.422761, -0.038140, -0.000100, 0.000000, -3.141593, 0.000000],accel_mss,speed_ms,0,blend_radius_m)
    |   movel(p[0.424123, -0.037198, -0.000100, 0.000000, -3.141593, 0.000000],accel_mss,speed_ms,0,blend_radius_m)
    |   movel(p[0.425365, -0.035753, -0.000100, 0.000000, -3.141593, 0.000000],accel_mss,speed_ms,0,blend_radius_m)
    |   movel(p[0.426399, -0.033924, -0.000100, 0.000000, 3.141593, 0.000000],accel_mss,speed_ms,0,blend_radius_m)
    |   movel(p[0.427144, -0.031836, -0.000100, 0.000000, -3.141593, 0.000000],accel_mss,speed_ms,0,blend_radius_m)
    |   movel(p[0.427378, -0.030620, -0.000100, 0.000000, -3.141593, 0.000000],accel_mss,speed_ms,0,blend_radius_m)
    |   movel(p[0.427482, -0.029158, -0.000100, 0.000000, -3.141593, 0.000000],accel_mss,speed_ms,0,blend_radius_m)
    |   movel(p[0.427458, -0.027773, -0.000100, 0.000000, -3.141593, 0.000000],accel_mss,speed_ms,0,blend_radius_m)
    |   movel(p[0.427276, -0.026853, -0.000100, 0.000000, 3.141593, 0.000000],accel_mss,speed_ms,0,blend_radius_m)
    |   movel(p[0.426502, -0.025075, -0.000100, 0.000000, 3.141593, 0.000000],accel_mss,speed_ms,0,blend_radius_m)
    |   movel(p[0.425512, -0.023629, -0.000100, 0.000000, -3.141593, 0.000000],accel_mss,speed_ms,0,blend_radius_m)
    |   movel(p[0.424255, -0.022460, -0.000100, 0.000000, -3.141593, 0.000000],accel_mss,speed_ms,0,blend_radius_m)
    |   movel(p[0.422686, -0.021510, -0.000100, 0.000000, -3.141593, 0.000000],accel_mss,speed_ms,0,blend_radius_m)
    |   movel(p[0.422011, -0.021182, -0.000100, 0.000000, -3.141593, 0.000000],accel_mss,speed_ms,0,blend_radius_m)
    |   movel(p[0.421336, -0.020853, -0.000100, 0.000000, -3.141593, 0.000000],accel_mss,speed_ms,0,blend_radius_m)
    |   movel(p[0.420211, -0.020856, -0.000100, 0.000000, 3.141593, 0.000000],accel_mss,speed_ms,0,blend_radius_m)
    |   movel(p[0.419086, -0.020859, -0.000100, 0.000000, -3.141593, 0.000000],accel_mss,speed_ms,0,blend_radius_m)
    |   movel(p[0.417935, -0.020875, -0.000100, 0.000000, -3.141593, 0.000000],accel_mss,speed_ms,0,blend_radius_m)
    |   movel(p[0.417122, -0.020921, -0.000100, 0.000000, 3.141593, 0.000000],accel_mss,speed_ms,0,blend_radius_m)
    |   movel(p[0.416491, -0.021003, -0.000100, 0.000000, 3.141593, 0.000000],accel_mss,speed_ms,0,blend_radius_m)
    |   movel(p[0.415936, -0.021135, -0.000100, 0.000000, 3.141593, 0.000000],accel_mss,speed_ms,0,blend_radius_m)
    |   movel(p[0.415109, -0.021418, -0.000100, 0.000000, -3.141593, 0.000000],accel_mss,speed_ms,0,blend_radius_m)
    |   movel(p[0.414297, -0.021761, -0.000100, 0.000000, 3.141593, 0.000000],accel_mss,speed_ms,0,blend_radius_m)
    |   movel(p[0.413614, -0.022105, -0.000100, 0.000000, -3.141593, 0.000000],accel_mss,speed_ms,0,blend_radius_m)
    |   movel(p[0.413308, -0.022357, -0.000100, 0.000000, -3.141593, 0.000000],accel_mss,speed_ms,0,0.000)
    |   movel(p[0.413225, -0.022442, -0.000100, 0.000000, -3.141593, 0.000000],accel_mss,speed_ms,0,0.000)
    |   movel(p[0.413130, -0.022513, -0.000100, 0.000000, 3.141593, 0.000000],accel_mss,speed_ms,0,0.000)
    |   movel(p[0.413035, -0.022563, -0.000100, 0.000000, 3.141593, 0.000000],accel_mss,speed_ms,0,0.000)
    |   movel(p[0.412712, -0.022678, -0.000100, 0.000000, -3.141593, 0.000000],accel_mss,speed_ms,0,0.000)
    |   movel(p[0.411704, -0.023664, -0.000100, 0.000000, -3.141593, 0.000000],accel_mss,speed_ms,0,blend_radius_m)
    |   movel(p[0.410711, -0.024664, -0.000100, 0.000000, -3.141593, 0.000000],accel_mss,speed_ms,0,blend_radius_m)
    |   movel(p[0.410611, -0.024909, -0.000100, 0.000000, -3.141593, 0.000000],accel_mss,speed_ms,0,0.000)
    |   movel(p[0.410479, -0.025151, -0.000100, 0.000000, -3.141593, 0.000000],accel_mss,speed_ms,0,0.000)
    |   movel(p[0.410333, -0.025326, -0.000100, 0.000000, -3.141593, 0.000000],accel_mss,speed_ms,0,0.000)
    |   movel(p[0.410161, -0.025503, -0.000100, 0.000000, -3.141593, 0.000000],accel_mss,speed_ms,0,0.000)
    |   movel(p[0.409989, -0.025678, -0.000100, 0.000000, -3.141593, 0.000000],accel_mss,speed_ms,0,0.000)
    |   movel(p[0.409843, -0.025847, -0.000100, 0.000000, -3.141593, 0.000000],accel_mss,speed_ms,0,0.000)
    |   movel(p[0.409734, -0.025994, -0.000100, 0.000000, -3.141593, 0.000000],accel_mss,speed_ms,0,0.000)
    |   movel(p[0.409689, -0.026150, -0.000100, 0.000000, -3.141593, 0.000000],accel_mss,speed_ms,0,0.000)
    |   movel(p[0.409568, -0.026347, -0.000100, 0.000000, -3.141593, 0.000000],accel_mss,speed_ms,0,0.000)
    |   movel(p[0.409410, -0.026579, -0.000100, 0.000000, 3.141593, 0.000000],accel_mss,speed_ms,0,0.000)
    |   movel(p[0.409223, -0.026828, -0.000100, 0.000000, -3.141593, 0.000000],accel_mss,speed_ms,0,0.000)
    |   movel(p[0.408829, -0.027348, -0.000100, 0.000000, -3.141593, 0.000000],accel_mss,speed_ms,0,blend_radius_m)
    |   movel(p[0.408564, -0.027736, -0.000100, 0.000000, -3.141593, 0.000000],accel_mss,speed_ms,0,0.000)
    |   movel(p[0.408371, -0.028074, -0.000100, 0.000000, -3.141593, 0.000000],accel_mss,speed_ms,0,0.000)
    |   movel(p[0.408211, -0.028428, -0.000100, 0.000000, -3.141593, 0.000000],accel_mss,speed_ms,0,0.000)
    |   movel(p[0.408141, -0.028594, -0.000100, 0.000000, -3.141593, 0.000000],accel_mss,speed_ms,0,0.000)
    |   movel(p[0.408054, -0.028781, -0.000100, 0.000000, -3.141593, 0.000000],accel_mss,speed_ms,0,0.000)
    |   movel(p[0.407965, -0.028962, -0.000100, 0.000000, -3.141593, 0.000000],accel_mss,speed_ms,0,0.000)
    |   movel(p[0.407887, -0.029103, -0.000100, 0.000000, 3.141593, 0.000000],accel_mss,speed_ms,0,0.000)
    |   movel(p[0.407396, -0.030047, -0.000100, 0.000000, -3.141593, 0.000000],accel_mss,speed_ms,0,blend_radius_m)
    |   movel(p[0.407013, -0.030989, -0.000100, 0.000000, 3.141593, 0.000000],accel_mss,speed_ms,0,blend_radius_m)
    |   movel(p[0.406646, -0.032178, -0.000100, 0.000000, -3.141593, 0.000000],accel_mss,speed_ms,0,blend_radius_m)
    |   movel(p[0.406185, -0.033978, -0.000100, 0.000000, -3.141593, 0.000000],accel_mss,speed_ms,0,blend_radius_m)
    |   movel(p[0.405691, -0.037126, -0.000100, 0.000000, -3.141593, 0.000000],accel_mss,speed_ms,0,blend_radius_m)
    |   # Splitting circular movement in 4 (instruction 1870:MoveC 1811)
    |   movel(p[0.405615, -0.038289, -0.000100, 0.000000, -3.141593, 0.000000],accel_mss,speed_ms,0,blend_radius_m)
    |   movel(p[0.405554, -0.039452, -0.000100, 0.000000, -3.141593, 0.000000],accel_mss,speed_ms,0,blend_radius_m)
    |   movel(p[0.405510, -0.040616, -0.000100, 0.000000, 3.141593, 0.000000],accel_mss,speed_ms,0,blend_radius_m)
    |   movel(p[0.405482, -0.041781, -0.000100, 0.000000, -3.141593, 0.000000],accel_mss,speed_ms,0,blend_radius_m)
    |   # Splitting circular movement in 4 (instruction 1871:MoveC 1812)
    |   movel(p[0.405470, -0.042997, -0.000100, 0.000000, -3.141593, 0.000000],accel_mss,speed_ms,0,blend_radius_m)
    |   movel(p[0.405476, -0.044213, -0.000100, 0.000000, 3.141593, 0.000000],accel_mss,speed_ms,0,blend_radius_m)
    |   movel(p[0.405499, -0.045429, -0.000100, 0.000000, 3.141593, 0.000000],accel_mss,speed_ms,0,blend_radius_m)
    |   movel(p[0.405539, -0.046645, -0.000100, 0.000000, 3.141593, 0.000000],accel_mss,speed_ms,0,blend_radius_m)
    |   # Splitting circular movement in 4 (instruction 1872:MoveC 1813)
    |   movel(p[0.405592, -0.047644, -0.000100, 0.000000, 3.141593, 0.000000],accel_mss,speed_ms,0,blend_radius_m)
    |   movel(p[0.405671, -0.048641, -0.000100, 0.000000, -3.141593, 0.000000],accel_mss,speed_ms,0,blend_radius_m)
    |   movel(p[0.405775, -0.049636, -0.000100, 0.000000, -3.141593, 0.000000],accel_mss,speed_ms,0,blend_radius_m)
    |   movel(p[0.405904, -0.050628, -0.000100, 0.000000, -3.141593, 0.000000],accel_mss,speed_ms,0,blend_radius_m)
    |   movel(p[0.406093, -0.051862, -0.000100, 0.000000, -3.141593, 0.000000],accel_mss,speed_ms,0,blend_radius_m)
    |   movel(p[0.406295, -0.053034, -0.000100, 0.000000, -3.141593, 0.000000],accel_mss,speed_ms,0,blend_radius_m)
    |   movel(p[0.406500, -0.054075, -0.000100, 0.000000, -3.141593, 0.000000],accel_mss,speed_ms,0,blend_radius_m)
    |   movel(p[0.406692, -0.054903, -0.000100, 0.000000, -3.141593, 0.000000],accel_mss,speed_ms,0,blend_radius_m)
    |   movel(p[0.406757, -0.055171, -0.000100, 0.000000, -3.141593, 0.000000],accel_mss,speed_ms,0,0.000)
    |   movel(p[0.406826, -0.055479, -0.000100, 0.000000, 3.141593, 0.000000],accel_mss,speed_ms,0,0.000)
    |   movel(p[0.406889, -0.055779, -0.000100, 0.000000, -3.141593, 0.000000],accel_mss,speed_ms,0,0.000)
